gfCNCPoint2[26382] = {X 371.8501, Y 39.8916, Z -3.8333, A 0.000, B 0.000, C 0.000 }
gfCNCPoint2[26383] = {X 370.5669, Y 42.1931, Z -3.8333, A 0.000, B 0.000, C 0.000 }
gfCNCPoint2[26384] = {X 369.0859, Y 44.3727, Z -3.8333, A 0.000, B 0.000, C 0.000 }
gfCNCPoint2[26385] = {X 368.9528, Y 44.5552, Z -3.8333, A 0.000, B 0.000, C 0.000 }
gfCNCPoint2[26386] = {X 368.8456, Y 44.6942, Z -3.8333, A 0.000, B 0.000, C 0.000 }
gfCNCPoint2[26387] = {X 368.1791, Y 45.5125, Z -3.8333, A 0.000, B 0.000, C 0.000 }
gfCNCPoint2[26388] = {X 366.6009, Y 47.2831, Z -3.8333, A 0.000, B 0.000, C 0.000 }
gfCNCPoint2[26389] = {X 364.8716, Y 48.9063, Z -3.8333, A 0.000, B 0.000, C 0.000 }
gfCNCPoint2[26390] = {X 363.0049, Y 50.3694, Z -3.8333, A 0.000, B 0.000, C 0.000 }
gfCNCPoint2[26391] = {X 361.0154, Y 51.6607, Z -3.8333, A 0.000, B 0.000, C 0.000 }
gfCNCPoint2[26392] = {X 358.9191, Y 52.7701, Z -3.8333, A 0.000, B 0.000, C 0.000 }
gfCNCPoint2[26393] = {X 358.4181, Y 53.0061, Z -3.8333, A 0.000, B 0.000, C 0.000 }
gfCNCPoint2[26394] = {X 356.2600, Y 53.8435, Z -3.8333, A 0.000, B 0.000, C 0.000 }
gfCNCPoint2[26395] = {X 354.0408, Y 54.5022, Z -3.8333, A 0.000, B 0.000, C 0.000 }
gfCNCPoint2[26396] = {X 351.7753, Y 54.9779, Z -3.8333, A 0.000, B 0.000, C 0.000 }
gfCNCPoint2[26397] = {X 349.4785, Y 55.2673, Z -3.8333, A 0.000, B 0.000, C 0.000 }
gfCNCPoint2[26398] = {X 347.1658, Y 55.3685, Z -3.8333, A 0.000, B 0.000, C 0.000 }
gfCNCPoint2[26399] = {X 344.5858, Y 55.3167, Z -3.8333, A 0.000, B 0.000, C 0.000 }
gfCNCPoint2[26400] = {X 342.0204, Y 55.0370, Z -3.8333, A 0.000, B 0.000, C 0.000 }
gfCNCPoint2[26401] = {X 339.4898, Y 54.5317, Z -3.8333, A 0.000, B 0.000, C 0.000 }
gfCNCPoint2[26402] = {X 337.0137, Y 53.8047, Z -3.8333, A 0.000, B 0.000, C 0.000 }
gfCNCPoint2[26403] = {X 334.7575, Y 52.9261, Z -3.8333, A 0.000, B 0.000, C 0.000 }
gfCNCPoint2[26404] = {X 332.5819, Y 51.8633, Z -3.8333, A 0.000, B 0.000, C 0.000 }
gfCNCPoint2[26405] = {X 331.5855, Y 51.2776, Z -3.8333, A 0.000, B 0.000, C 0.000 }
gfCNCPoint2[26406] = {X 330.6132, Y 50.6529, Z -3.8333, A 0.000, B 0.000, C 0.000 }
gfCNCPoint2[26407] = {X 331.5791, Y 51.6068, Z -3.8333, A 0.000, B 0.000, C 0.000 }
gfCNCPoint2[26408] = {X 332.4020, Y 52.6865, Z -3.8333, A 0.000, B 0.000, C 0.000 }
gfCNCPoint2[26409] = {X 333.0657, Y 53.8706, Z -3.8333, A 0.000, B 0.000, C 0.000 }
gfCNCPoint2[26410] = {X 333.5573, Y 55.1360, Z -3.8333, A 0.000, B 0.000, C 0.000 }
gfCNCPoint2[26411] = {X 333.8670, Y 56.4577, Z -3.8333, A 0.000, B 0.000, C 0.000 }
gfCNCPoint2[26412] = {X 333.9597, Y 57.2264, Z -3.8333, A 0.000, B 0.000, C 0.000 }
gfCNCPoint2[26413] = {X 333.9907, Y 58.0000, Z -3.8333, A 0.000, B 0.000, C 0.000 }
gfCNCPoint2[26414] = {X 333.9906, Y 58.9572, Z -3.8333, A 0.000, B 0.000, C 0.000 }
gfCNCPoint2[26415] = {X 333.8743, Y 60.4101, Z -3.8333, A 0.000, B 0.000, C 0.000 }
gfCNCPoint2[26416] = {X 333.5421, Y 61.8292, Z -3.8333, A 0.000, B 0.000, C 0.000 }
gfCNCPoint2[26417] = {X 333.0014, Y 63.1827, Z -3.8333, A 0.000, B 0.000, C 0.000 }
gfCNCPoint2[26418] = {X 332.2643, Y 64.4401, Z -3.8333, A 0.000, B 0.000, C 0.000 }
gfCNCPoint2[26419] = {X 331.3475, Y 65.5731, Z -3.8333, A 0.000, B 0.000, C 0.000 }
gfCNCPoint2[26420] = {X 330.2716, Y 66.5563, Z -3.8333, A 0.000, B 0.000, C 0.000 }
gfCNCPoint2[26421] = {X 330.2729, Y 83.2032, Z -3.8333, A 0.000, B 0.000, C 0.000 }
gfCNCPoint2[26422] = {X 330.2766, Y 83.5831, Z -3.8333, A 0.000, B 0.000, C 0.000 }
gfCNCPoint2[26423] = {X 330.3838, Y 83.6086, Z -3.8333, A 0.000, B 0.000, C 0.000 }
gfCNCPoint2[26424] = {X 333.0907, Y 84.1513, Z -3.8333, A 0.000, B 0.000, C 0.000 }
gfCNCPoint2[26425] = {X 335.8298, Y 84.4970, Z -3.8333, A 0.000, B 0.000, C 0.000 }
gfCNCPoint2[26426] = {X 339.8061, Y 84.8050, Z -3.8333, A 0.000, B 0.000, C 0.000 }
gfCNCPoint2[26427] = {X 343.7906, Y 84.9773, Z -3.8333, A 0.000, B 0.000, C 0.000 }
gfCNCPoint2[26428] = {X 347.7787, Y 85.0135, Z -3.8333, A 0.000, B 0.000, C 0.000 }
gfCNCPoint2[26429] = {X 351.9888, Y 84.9781, Z -3.8333, A 0.000, B 0.000, C 0.000 }
gfCNCPoint2[26430] = {X 356.1949, Y 84.7906, Z -3.8333, A 0.000, B 0.000, C 0.000 }
gfCNCPoint2[26431] = {X 360.3914, Y 84.4512, Z -3.8333, A 0.000, B 0.000, C 0.000 }
gfCNCPoint2[26432] = {X 362.9935, Y 84.1044, Z -3.8333, A 0.000, B 0.000, C 0.000 }
gfCNCPoint2[26433] = {X 365.5604, Y 83.5544, Z -3.8333, A 0.000, B 0.000, C 0.000 }
gfCNCPoint2[26434] = {X 365.5591, Y 66.5616, Z -3.8333, A 0.000, B 0.000, C 0.000 }
gfCNCPoint2[26435] = {X 364.4966, Y 65.5962, Z -3.8333, A 0.000, B 0.000, C 0.000 }
gfCNCPoint2[26436] = {X 363.5885, Y 64.4843, Z -3.8333, A 0.000, B 0.000, C 0.000 }
gfCNCPoint2[26437] = {X 362.8549, Y 63.2504, Z -3.8333, A 0.000, B 0.000, C 0.000 }
gfCNCPoint2[26438] = {X 349.9657, Y 69.6713, Z -3.8333, A 0.000, B 0.000, C 0.000 }
gfCNCPoint2[26439] = {X 348.6643, Y 69.7393, Z -3.8333, A 0.000, B 0.000, C 0.000 }
gfCNCPoint2[26440] = {X 347.3614, Y 69.7677, Z -3.8333, A 0.000, B 0.000, C 0.000 }
gfCNCPoint2[26441] = {X 346.5840, Y 69.7768, Z -3.8333, A 0.000, B 0.000, C 0.000 }
gfCNCPoint2[26442] = {X 345.8066, Y 69.7721, Z -3.8333, A 0.000, B 0.000, C 0.000 }
gfCNCPoint2[26443] = {X 345.5899, Y 70.1915, Z -3.8333, A 0.000, B 0.000, C 0.000 }
gfCNCPoint2[26444] = {X 345.3650, Y 70.6066, Z -3.8333, A 0.000, B 0.000, C 0.000 }
gfCNCPoint2[26445] = {X 346.5779, Y 70.6169, Z -3.8333, A 0.000, B 0.000, C 0.000 }
gfCNCPoint2[26446] = {X 347.7907, Y 70.6129, Z -3.8333, A 0.000, B 0.000, C 0.000 }
gfCNCPoint2[26447] = {X 349.1243, Y 70.6187, Z -3.8333, A 0.000, B 0.000, C 0.000 }
gfCNCPoint2[26448] = {X 350.4578, Y 70.6071, Z -3.8333, A 0.000, B 0.000, C 0.000 }
gfCNCPoint2[26449] = {X 350.2066, Y 70.1419, Z -3.8333, A 0.000, B 0.000, C 0.000 }
gfCNCPoint2[26450] = {X 349.9657, Y 69.6713, Z -3.8333, A 0.000, B 0.000, C 0.000 }
gfCNCPoint2[26451] = {X 352.1139, Y 68.6012, Z -3.8333, A 0.000, B 0.000, C 0.000 }
gfCNCPoint2[26452] = {X 351.7677, Y 67.8727, Z -3.8333, A 0.000, B 0.000, C 0.000 }
gfCNCPoint2[26453] = {X 351.4489, Y 67.1318, Z -3.8333, A 0.000, B 0.000, C 0.000 }
gfCNCPoint2[26454] = {X 349.3919, Y 67.3025, Z -3.8333, A 0.000, B 0.000, C 0.000 }
gfCNCPoint2[26455] = {X 347.3288, Y 67.3678, Z -3.8333, A 0.000, B 0.000, C 0.000 }
gfCNCPoint2[26456] = {X 345.8122, Y 67.3719, Z -3.8333, A 0.000, B 0.000, C 0.000 }
gfCNCPoint2[26457] = {X 344.2965, Y 67.3201, Z -3.8333, A 0.000, B 0.000, C 0.000 }
gfCNCPoint2[26458] = {X 343.8102, Y 68.3954, Z -3.8333, A 0.000, B 0.000, C 0.000 }
gfCNCPoint2[26459] = {X 343.2661, Y 69.4427, Z -3.8333, A 0.000, B 0.000, C 0.000 }
gfCNCPoint2[26460] = {X 342.7868, Y 70.2642, Z -3.8333, A 0.000, B 0.000, C 0.000 }
gfCNCPoint2[26461] = {X 342.2719, Y 71.0639, Z -3.8333, A 0.000, B 0.000, C 0.000 }
gfCNCPoint2[26462] = {X 342.2721, Y 72.9175, Z -3.8333, A 0.000, B 0.000, C 0.000 }
gfCNCPoint2[26463] = {X 343.8009, Y 72.9730, Z -3.8333, A 0.000, B 0.000, C 0.000 }
gfCNCPoint2[26464] = {X 345.3303, Y 73.0063, Z -3.8333, A 0.000, B 0.000, C 0.000 }
gfCNCPoint2[26465] = {X 346.5595, Y 73.0169, Z -3.8333, A 0.000, B 0.000, C 0.000 }
gfCNCPoint2[26466] = {X 347.7887, Y 73.0130, Z -3.8333, A 0.000, B 0.000, C 0.000 }
gfCNCPoint2[26467] = {X 349.1416, Y 73.0187, Z -3.8333, A 0.000, B 0.000, C 0.000 }
gfCNCPoint2[26468] = {X 350.4943, Y 73.0069, Z -3.8333, A 0.000, B 0.000, C 0.000 }
gfCNCPoint2[26469] = {X 352.0273, Y 72.9723, Z -3.8333, A 0.000, B 0.000, C 0.000 }
gfCNCPoint2[26470] = {X 353.5596, Y 72.9152, Z -3.8333, A 0.000, B 0.000, C 0.000 }
gfCNCPoint2[26471] = {X 353.5595, Y 71.0777, Z -3.8333, A 0.000, B 0.000, C 0.000 }
gfCNCPoint2[26472] = {X 353.0401, Y 70.2718, Z -3.8333, A 0.000, B 0.000, C 0.000 }
gfCNCPoint2[26473] = {X 352.5569, Y 69.4437, Z -3.8333, A 0.000, B 0.000, C 0.000 }
gfCNCPoint2[26474] = {X 352.3308, Y 69.0249, Z -3.8333, A 0.000, B 0.000, C 0.000 }
gfCNCPoint2[26475] = {X 352.1139, Y 68.6012, Z -3.8333, A 0.000, B 0.000, C 0.000 }
gfCNCPoint2[26476] = {X 354.2621, Y 67.5310, Z -3.8333, A 0.000, B 0.000, C 0.000 }
gfCNCPoint2[26477] = {X 353.5960, Y 66.0387, Z -3.8333, A 0.000, B 0.000, C 0.000 }
gfCNCPoint2[26478] = {X 353.0588, Y 64.4954, Z -3.8333, A 0.000, B 0.000, C 0.000 }
gfCNCPoint2[26479] = {X 350.1865, Y 64.8415, Z -3.8333, A 0.000, B 0.000, C 0.000 }
gfCNCPoint2[26480] = {X 347.2961, Y 64.9680, Z -3.8333, A 0.000, B 0.000, C 0.000 }
gfCNCPoint2[26481] = {X 344.9823, Y 64.9488, Z -3.8333, A 0.000, B 0.000, C 0.000 }
gfCNCPoint2[26482] = {X 342.6738, Y 64.7916, Z -3.8333, A 0.000, B 0.000, C 0.000 }
gfCNCPoint2[26483] = {X 341.9390, Y 66.7265, Z -3.8333, A 0.000, B 0.000, C 0.000 }
gfCNCPoint2[26484] = {X 341.0015, Y 68.5717, Z -3.8333, A 0.000, B 0.000, C 0.000 }
gfCNCPoint2[26485] = {X 339.8719, Y 70.3060, Z -3.8333, A 0.000, B 0.000, C 0.000 }
gfCNCPoint2[26486] = {X 339.8723, Y 75.1904, Z -3.8333, A 0.000, B 0.000, C 0.000 }
gfCNCPoint2[26487] = {X 343.8274, Y 75.3748, Z -3.8333, A 0.000, B 0.000, C 0.000 }
gfCNCPoint2[26488] = {X 347.7867, Y 75.4132, Z -3.8333, A 0.000, B 0.000, C 0.000 }
gfCNCPoint2[26489] = {X 351.8754, Y 75.3776, Z -3.8333, A 0.000, B 0.000, C 0.000 }
gfCNCPoint2[26490] = {X 355.9598, Y 75.1858, Z -3.8333, A 0.000, B 0.000, C 0.000 }
gfCNCPoint2[26491] = {X 355.9594, Y 70.3187, Z -3.8333, A 0.000, B 0.000, C 0.000 }
gfCNCPoint2[26492] = {X 355.0517, Y 68.9608, Z -3.8333, A 0.000, B 0.000, C 0.000 }
gfCNCPoint2[26493] = {X 354.2621, Y 67.5310, Z -3.8333, A 0.000, B 0.000, C 0.000 }
gfCNCPoint2[26494] = {X 356.4103, Y 66.4608, Z -3.8333, A 0.000, B 0.000, C 0.000 }
gfCNCPoint2[26495] = {X 355.7399, Y 64.9296, Z -3.8333, A 0.000, B 0.000, C 0.000 }
gfCNCPoint2[26496] = {X 355.2243, Y 63.3395, Z -3.8333, A 0.000, B 0.000, C 0.000 }
gfCNCPoint2[26497] = {X 354.8685, Y 61.7062, Z -3.8333, A 0.000, B 0.000, C 0.000 }
gfCNCPoint2[26498] = {X 352.3563, Y 62.1755, Z -3.8333, A 0.000, B 0.000, C 0.000 }
gfCNCPoint2[26499] = {X 349.8170, Y 62.4634, Z -3.8333, A 0.000, B 0.000, C 0.000 }
gfCNCPoint2[26500] = {X 347.2635, Y 62.5681, Z -3.8333, A 0.000, B 0.000, C 0.000 }
gfCNCPoint2[26501] = {X 345.1281, Y 62.5526, Z -3.8333, A 0.000, B 0.000, C 0.000 }
gfCNCPoint2[26502] = {X 342.9973, Y 62.4117, Z -3.8333, A 0.000, B 0.000, C 0.000 }
gfCNCPoint2[26503] = {X 340.8785, Y 62.1460, Z -3.8333, A 0.000, B 0.000, C 0.000 }
gfCNCPoint2[26504] = {X 340.4886, Y 63.7339, Z -3.8333, A 0.000, B 0.000, C 0.000 }
gfCNCPoint2[26505] = {X 339.9473, Y 65.2768, Z -3.8333, A 0.000, B 0.000, C 0.000 }
gfCNCPoint2[26506] = {X 339.2595, Y 66.7602, Z -3.8333, A 0.000, B 0.000, C 0.000 }
gfCNCPoint2[26507] = {X 338.4318, Y 68.1703, Z -3.8333, A 0.000, B 0.000, C 0.000 }
gfCNCPoint2[26508] = {X 337.4718, Y 69.4939, Z -3.8333, A 0.000, B 0.000, C 0.000 }
gfCNCPoint2[26509] = {X 337.4724, Y 77.4160, Z -3.8333, A 0.000, B 0.000, C 0.000 }
gfCNCPoint2[26510] = {X 340.9052, Y 77.6563, Z -3.8333, A 0.000, B 0.000, C 0.000 }
gfCNCPoint2[26511] = {X 344.3437, Y 77.7887, Z -3.8333, A 0.000, B 0.000, C 0.000 }
gfCNCPoint2[26512] = {X 347.7847, Y 77.8133, Z -3.8333, A 0.000, B 0.000, C 0.000 }
gfCNCPoint2[26513] = {X 351.3135, Y 77.7924, Z -3.8333, A 0.000, B 0.000, C 0.000 }
gfCNCPoint2[26514] = {X 354.8398, Y 77.6576, Z -3.8333, A 0.000, B 0.000, C 0.000 }
gfCNCPoint2[26515] = {X 358.3599, Y 77.4091, Z -3.8333, A 0.000, B 0.000, C 0.000 }
gfCNCPoint2[26516] = {X 358.3594, Y 69.5053, Z -3.8333, A 0.000, B 0.000, C 0.000 }
gfCNCPoint2[26517] = {X 357.3031, Y 68.0354, Z -3.8333, A 0.000, B 0.000, C 0.000 }
gfCNCPoint2[26518] = {X 356.4103, Y 66.4608, Z -3.8333, A 0.000, B 0.000, C 0.000 }
gfCNCPoint2[26519] = {X 358.5585, Y 65.3907, Z -3.8333, A 0.000, B 0.000, C 0.000 }
gfCNCPoint2[26520] = {X 357.9834, Y 64.0771, Z -3.8333, A 0.000, B 0.000, C 0.000 }
gfCNCPoint2[26521] = {X 357.5411, Y 62.7131, Z -3.8333, A 0.000, B 0.000, C 0.000 }
gfCNCPoint2[26522] = {X 357.2359, Y 61.3120, Z -3.8333, A 0.000, B 0.000, C 0.000 }
gfCNCPoint2[26523] = {X 357.0916, Y 60.1636, Z -3.8333, A 0.000, B 0.000, C 0.000 }
gfCNCPoint2[26524] = {X 357.0395, Y 59.0073, Z -3.8333, A 0.000, B 0.000, C 0.000 }
gfCNCPoint2[26525] = {X 357.0394, Y 58.6392, Z -3.8333, A 0.000, B 0.000, C 0.000 }
gfCNCPoint2[26526] = {X 355.6989, Y 59.0302, Z -3.8333, A 0.000, B 0.000, C 0.000 }
gfCNCPoint2[26527] = {X 354.3432, Y 59.3643, Z -3.8333, A 0.000, B 0.000, C 0.000 }
gfCNCPoint2[26528] = {X 351.9938, Y 59.8031, Z -3.8333, A 0.000, B 0.000, C 0.000 }
gfCNCPoint2[26529] = {X 349.6190, Y 60.0715, Z -3.8333, A 0.000, B 0.000, C 0.000 }
gfCNCPoint2[26530] = {X 347.2310, Y 60.1683, Z -3.8333, A 0.000, B 0.000, C 0.000 }
gfCNCPoint2[26531] = {X 344.3949, Y 60.1141, Z -3.8333, A 0.000, B 0.000, C 0.000 }
gfCNCPoint2[26532] = {X 341.5732, Y 59.8235, Z -3.8333, A 0.000, B 0.000, C 0.000 }
gfCNCPoint2[26533] = {X 338.7856, Y 59.2985, Z -3.8333, A 0.000, B 0.000, C 0.000 }
gfCNCPoint2[26534] = {X 338.6399, Y 60.9979, Z -3.8333, A 0.000, B 0.000, C 0.000 }
gfCNCPoint2[26535] = {X 338.2960, Y 62.6684, Z -3.8333, A 0.000, B 0.000, C 0.000 }
gfCNCPoint2[26536] = {X 337.7585, Y 64.2871, Z -3.8333, A 0.000, B 0.000, C 0.000 }
gfCNCPoint2[26537] = {X 337.0349, Y 65.8316, Z -3.8333, A 0.000, B 0.000, C 0.000 }
gfCNCPoint2[26538] = {X 336.1352, Y 67.2806, Z -3.8333, A 0.000, B 0.000, C 0.000 }
gfCNCPoint2[26539] = {X 335.0717, Y 68.6140, Z -3.8333, A 0.000, B 0.000, C 0.000 }
gfCNCPoint2[26540] = {X 335.0726, Y 79.5885, Z -3.8333, A 0.000, B 0.000, C 0.000 }
gfCNCPoint2[26541] = {X 335.6679, Y 79.6579, Z -3.8333, A 0.000, B 0.000, C 0.000 }
gfCNCPoint2[26542] = {X 336.2643, Y 79.7167, Z -3.8333, A 0.000, B 0.000, C 0.000 }
gfCNCPoint2[26543] = {X 340.0974, Y 80.0139, Z -3.8333, A 0.000, B 0.000, C 0.000 }
gfCNCPoint2[26544] = {X 343.9383, Y 80.1795, Z -3.8333, A 0.000, B 0.000, C 0.000 }
gfCNCPoint2[26545] = {X 347.7827, Y 80.2134, Z -3.8333, A 0.000, B 0.000, C 0.000 }
gfCNCPoint2[26546] = {X 351.8380, Y 80.1804, Z -3.8333, A 0.000, B 0.000, C 0.000 }
gfCNCPoint2[26547] = {X 355.8894, Y 80.0003, Z -3.8333, A 0.000, B 0.000, C 0.000 }
gfCNCPoint2[26548] = {X 359.9315, Y 79.6733, Z -3.8333, A 0.000, B 0.000, C 0.000 }
gfCNCPoint2[26549] = {X 360.3461, Y 79.6317, Z -3.8333, A 0.000, B 0.000, C 0.000 }
gfCNCPoint2[26550] = {X 360.7601, Y 79.5840, Z -3.8333, A 0.000, B 0.000, C 0.000 }
gfCNCPoint2[26551] = {X 360.7593, Y 68.6239, Z -3.8333, A 0.000, B 0.000, C 0.000 }
gfCNCPoint2[26552] = {X 359.9292, Y 67.6140, Z -3.8333, A 0.000, B 0.000, C 0.000 }
gfCNCPoint2[26553] = {X 359.1936, Y 66.5333, Z -3.8333, A 0.000, B 0.000, C 0.000 }
gfCNCPoint2[26554] = {X 358.5585, Y 65.3907, Z -3.8333, A 0.000, B 0.000, C 0.000 }
gfCNCPoint2[26555] = {X 360.7067, Y 64.3205, Z -3.8333, A 0.000, B 0.000, C 0.000 }
gfCNCPoint2[26556] = {X 360.1634, Y 63.0537, Z -3.8333, A 0.000, B 0.000, C 0.000 }
gfCNCPoint2[26557] = {X 359.7680, Y 61.7332, Z -3.8333, A 0.000, B 0.000, C 0.000 }
gfCNCPoint2[26558] = {X 359.5257, Y 60.3762, Z -3.8333, A 0.000, B 0.000, C 0.000 }
gfCNCPoint2[26559] = {X 359.4395, Y 59.0005, Z -3.8333, A 0.000, B 0.000, C 0.000 }
gfCNCPoint2[26560] = {X 359.4393, Y 58.0000, Z -3.8333, A 0.000, B 0.000, C 0.000 }
gfCNCPoint2[26561] = {X 359.5343, Y 56.4880, Z -3.8333, A 0.000, B 0.000, C 0.000 }
gfCNCPoint2[26562] = {X 359.8178, Y 54.9997, Z -3.8333, A 0.000, B 0.000, C 0.000 }
gfCNCPoint2[26563] = {X 359.4090, Y 55.1923, Z -3.8333, A 0.000, B 0.000, C 0.000 }
gfCNCPoint2[26564] = {X 357.8796, Y 55.8125, Z -3.8333, A 0.000, B 0.000, C 0.000 }
gfCNCPoint2[26565] = {X 356.3191, Y 56.3499, Z -3.8333, A 0.000, B 0.000, C 0.000 }
gfCNCPoint2[26566] = {X 354.0855, Y 56.9613, Z -3.8333, A 0.000, B 0.000, C 0.000 }
gfCNCPoint2[26567] = {X 351.8122, Y 57.4030, Z -3.8333, A 0.000, B 0.000, C 0.000 }
gfCNCPoint2[26568] = {X 349.5122, Y 57.6725, Z -3.8333, A 0.000, B 0.000, C 0.000 }
gfCNCPoint2[26569] = {X 347.1984, Y 57.7684, Z -3.8333, A 0.000, B 0.000, C 0.000 }
gfCNCPoint2[26570] = {X 344.5554, Y 57.7194, Z -3.8333, A 0.000, B 0.000, C 0.000 }
gfCNCPoint2[26571] = {X 341.9257, Y 57.4495, Z -3.8333, A 0.000, B 0.000, C 0.000 }
gfCNCPoint2[26572] = {X 339.3279, Y 56.9606, Z -3.8333, A 0.000, B 0.000, C 0.000 }
gfCNCPoint2[26573] = {X 337.7708, Y 56.5573, Z -3.8333, A 0.000, B 0.000, C 0.000 }
gfCNCPoint2[26574] = {X 336.2364, Y 56.0753, Z -3.8333, A 0.000, B 0.000, C 0.000 }
gfCNCPoint2[26575] = {X 336.3520, Y 57.0346, Z -3.8333, A 0.000, B 0.000, C 0.000 }
gfCNCPoint2[26576] = {X 336.3907, Y 58.0000, Z -3.8333, A 0.000, B 0.000, C 0.000 }
gfCNCPoint2[26577] = {X 336.3906, Y 58.9688, Z -3.8333, A 0.000, B 0.000, C 0.000 }
gfCNCPoint2[26578] = {X 336.3892, Y 59.1016, Z -3.8333, A 0.000, B 0.000, C 0.000 }
gfCNCPoint2[26579] = {X 336.3864, Y 59.2343, Z -3.8333, A 0.000, B 0.000, C 0.000 }
gfCNCPoint2[26580] = {X 336.2427, Y 60.7986, Z -3.8333, A 0.000, B 0.000, C 0.000 }
gfCNCPoint2[26581] = {X 335.8980, Y 62.3311, Z -3.8333, A 0.000, B 0.000, C 0.000 }
gfCNCPoint2[26582] = {X 335.3578, Y 63.8062, Z -3.8333, A 0.000, B 0.000, C 0.000 }
gfCNCPoint2[26583] = {X 334.6315, Y 65.1990, Z -3.8333, A 0.000, B 0.000, C 0.000 }
gfCNCPoint2[26584] = {X 333.7310, Y 66.4861, Z -3.8333, A 0.000, B 0.000, C 0.000 }
gfCNCPoint2[26585] = {X 332.6717, Y 67.6460, Z -3.8333, A 0.000, B 0.000, C 0.000 }
gfCNCPoint2[26586] = {X 332.6728, Y 81.6420, Z -3.8333, A 0.000, B 0.000, C 0.000 }
gfCNCPoint2[26587] = {X 334.3529, Y 81.9144, Z -3.8333, A 0.000, B 0.000, C 0.000 }
gfCNCPoint2[26588] = {X 336.0440, Y 82.1065, Z -3.8333, A 0.000, B 0.000, C 0.000 }
gfCNCPoint2[26589] = {X 339.9497, Y 82.4094, Z -3.8333, A 0.000, B 0.000, C 0.000 }
gfCNCPoint2[26590] = {X 343.8635, Y 82.5784, Z -3.8333, A 0.000, B 0.000, C 0.000 }
gfCNCPoint2[26591] = {X 347.7807, Y 82.6135, Z -3.8333, A 0.000, B 0.000, C 0.000 }
gfCNCPoint2[26592] = {X 351.9134, Y 82.5792, Z -3.8333, A 0.000, B 0.000, C 0.000 }
gfCNCPoint2[26593] = {X 356.0420, Y 82.3954, Z -3.8333, A 0.000, B 0.000, C 0.000 }
gfCNCPoint2[26594] = {X 360.1614, Y 82.0623, Z -3.8333, A 0.000, B 0.000, C 0.000 }
gfCNCPoint2[26595] = {X 361.6660, Y 81.8847, Z -3.8333, A 0.000, B 0.000, C 0.000 }
gfCNCPoint2[26596] = {X 363.1603, Y 81.6340, Z -3.8333, A 0.000, B 0.000, C 0.000 }
gfCNCPoint2[26597] = {X 363.1592, Y 67.6539, Z -3.8333, A 0.000, B 0.000, C 0.000 }
gfCNCPoint2[26598] = {X 362.2157, Y 66.6393, Z -3.8333, A 0.000, B 0.000, C 0.000 }
gfCNCPoint2[26599] = {X 361.3946, Y 65.5232, Z -3.8333, A 0.000, B 0.000, C 0.000 }
gfCNCPoint2[26600] = {X 360.7067, Y 64.3205, Z -3.8333, A 0.000, B 0.000, C 0.000 }
gfCNCPoint2[26601] = {X 362.8549, Y 63.2504, Z -3.8333, A 0.000, B 0.000, C 0.000 }
gfCNCPoint2[26602] = {X 362.3011, Y 61.8884, Z -3.8333, A 0.000, B 0.000, C 0.000 }
gfCNCPoint2[26603] = {X 361.9600, Y 60.4583, Z -3.8333, A 0.000, B 0.000, C 0.000 }
gfCNCPoint2[26604] = {X 361.8395, Y 58.9930, Z -3.8333, A 0.000, B 0.000, C 0.000 }
gfCNCPoint2[26605] = {X 361.8393, Y 58.0000, Z -3.8333, A 0.000, B 0.000, C 0.000 }
gfCNCPoint2[26606] = {X 361.9154, Y 56.7884, Z -3.8333, A 0.000, B 0.000, C 0.000 }
gfCNCPoint2[26607] = {X 362.1426, Y 55.5958, Z -3.8333, A 0.000, B 0.000, C 0.000 }
gfCNCPoint2[26608] = {X 362.5739, Y 54.3010, Z -3.8333, A 0.000, B 0.000, C 0.000 }
gfCNCPoint2[26609] = {X 363.1830, Y 53.0798, Z -3.8333, A 0.000, B 0.000, C 0.000 }
gfCNCPoint2[26610] = {X 363.9578, Y 51.9563, Z -3.8333, A 0.000, B 0.000, C 0.000 }
gfCNCPoint2[26611] = {X 364.8829, Y 50.9530, Z -3.8333, A 0.000, B 0.000, C 0.000 }
gfCNCPoint2[26612] = {X 365.9399, Y 50.0897, Z -3.8333, A 0.000, B 0.000, C 0.000 }
gfCNCPoint2[26613] = {X 367.1078, Y 49.3837, Z -3.8333, A 0.000, B 0.000, C 0.000 }
gfCNCPoint2[26614] = {X 368.3634, Y 48.8489, Z -3.8333, A 0.000, B 0.000, C 0.000 }
gfCNCPoint2[26615] = {X 369.6818, Y 48.4960, Z -3.8333, A 0.000, B 0.000, C 0.000 }
gfCNCPoint2[26616] = {X 371.0366, Y 48.3320, Z -3.8333, A 0.000, B 0.000, C 0.000 }
gfCNCPoint2[26617] = {X 371.2779, Y 48.3230, Z -3.8333, A 0.000, B 0.000, C 0.000 }
gfCNCPoint2[26618] = {X 371.5193, Y 48.3200, Z -3.8333, A 0.000, B 0.000, C 0.000 }
gfCNCPoint2[26619] = {X 388.0597, Y 48.3200, Z -3.8333, A 0.000, B 0.000, C 0.000 }
gfCNCPoint2[26620] = {X 389.4419, Y 48.4192, Z -3.8333, A 0.000, B 0.000, C 0.000 }
gfCNCPoint2[26621] = {X 390.7958, Y 48.7147, Z -3.8333, A 0.000, B 0.000, C 0.000 }
gfCNCPoint2[26622] = {X 392.0936, Y 49.2006, Z -3.8333, A 0.000, B 0.000, C 0.000 }
gfCNCPoint2[26623] = {X 393.3087, Y 49.8667, Z -3.8333, A 0.000, B 0.000, C 0.000 }
gfCNCPoint2[26624] = {X 394.5333, Y 49.1962, Z -3.8333, A 0.000, B 0.000, C 0.000 }
gfCNCPoint2[26625] = {X 395.8416, Y 48.7089, Z -3.8333, A 0.000, B 0.000, C 0.000 }
gfCNCPoint2[26626] = {X 397.1858, Y 48.4177, Z -3.8333, A 0.000, B 0.000, C 0.000 }
gfCNCPoint2[26627] = {X 398.5577, Y 48.3200, Z -3.8333, A 0.000, B 0.000, C 0.000 }
gfCNCPoint2[26628] = {X 398.7346, Y 48.3200, Z -3.8333, A 0.000, B 0.000, C 0.000 }
gfCNCPoint2[26629] = {X 398.1859, Y 47.6069, Z -3.8333, A 0.000, B 0.000, C 0.000 }
gfCNCPoint2[26630] = {X 397.7774, Y 46.8051, Z -3.8333, A 0.000, B 0.000, C 0.000 }
gfCNCPoint2[26631] = {X 397.5230, Y 45.9420, Z -3.8333, A 0.000, B 0.000, C 0.000 }
gfCNCPoint2[26632] = {X 397.4561, Y 45.4921, Z -3.8333, A 0.000, B 0.000, C 0.000 }
gfCNCPoint2[26633] = {X 397.4314, Y 45.0378, Z -3.8333, A 0.000, B 0.000, C 0.000 }
gfCNCPoint2[26634] = {X 397.4316, Y 44.1456, Z -3.8333, A 0.000, B 0.000, C 0.000 }
gfCNCPoint2[26635] = {X 397.5413, Y 43.1780, Z -3.8333, A 0.000, B 0.000, C 0.000 }
gfCNCPoint2[26636] = {X 397.8410, Y 42.2514, Z -3.8333, A 0.000, B 0.000, C 0.000 }
gfCNCPoint2[26637] = {X 398.3186, Y 41.4029, Z -3.8333, A 0.000, B 0.000, C 0.000 }
gfCNCPoint2[26638] = {X 398.9552, Y 40.6660, Z -3.8333, A 0.000, B 0.000, C 0.000 }
gfCNCPoint2[26639] = {X 398.9552, Y 31.8228, Z -3.8333, A 0.000, B 0.000, C 0.000 }
gfCNCPoint2[26640] = {X 396.7500, Y 27.9882, Z -3.8333, A 0.000, B 0.000, C 0.000 }
gfCNCPoint2[26641] = {X 386.3474, Y 33.9703, Z -3.8333, A 0.000, B 0.000, C 0.000 }
gfCNCPoint2[26642] = {X 386.2664, Y 34.3979, Z -3.8333, A 0.000, B 0.000, C 0.000 }
gfCNCPoint2[26643] = {X 386.1817, Y 34.8247, Z -3.8333, A 0.000, B 0.000, C 0.000 }
gfCNCPoint2[26644] = {X 386.0227, Y 35.5739, Z -3.8333, A 0.000, B 0.000, C 0.000 }
gfCNCPoint2[26645] = {X 385.8500, Y 36.3200, Z -3.8333, A 0.000, B 0.000, C 0.000 }
gfCNCPoint2[26646] = {X 386.9552, Y 36.3200, Z -3.8333, A 0.000, B 0.000, C 0.000 }
gfCNCPoint2[26647] = {X 386.9552, Y 35.0272, Z -3.8333, A 0.000, B 0.000, C 0.000 }
gfCNCPoint2[26648] = {X 386.3474, Y 33.9703, Z -3.8333, A 0.000, B 0.000, C 0.000 }
gfCNCPoint2[26649] = {X 388.4279, Y 32.7739, Z -3.8333, A 0.000, B 0.000, C 0.000 }
gfCNCPoint2[26650] = {X 384.7446, Y 26.3688, Z -3.8333, A 0.000, B 0.000, C 0.000 }
gfCNCPoint2[26651] = {X 384.6157, Y 28.7693, Z -3.8333, A 0.000, B 0.000, C 0.000 }
gfCNCPoint2[26652] = {X 384.3630, Y 31.1599, Z -3.8333, A 0.000, B 0.000, C 0.000 }
gfCNCPoint2[26653] = {X 383.9874, Y 33.5342, Z -3.8333, A 0.000, B 0.000, C 0.000 }
gfCNCPoint2[26654] = {X 383.9103, Y 33.9411, Z -3.8333, A 0.000, B 0.000, C 0.000 }
gfCNCPoint2[26655] = {X 383.8296, Y 34.3474, Z -3.8333, A 0.000, B 0.000, C 0.000 }
gfCNCPoint2[26656] = {X 383.6797, Y 35.0539, Z -3.8333, A 0.000, B 0.000, C 0.000 }
gfCNCPoint2[26657] = {X 383.5169, Y 35.7576, Z -3.8333, A 0.000, B 0.000, C 0.000 }
gfCNCPoint2[26658] = {X 383.1270, Y 37.2469, Z -3.8333, A 0.000, B 0.000, C 0.000 }
gfCNCPoint2[26659] = {X 382.6793, Y 38.7200, Z -3.8333, A 0.000, B 0.000, C 0.000 }
gfCNCPoint2[26660] = {X 388.0597, Y 38.7200, Z -3.8333, A 0.000, B 0.000, C 0.000 }
gfCNCPoint2[26661] = {X 388.4821, Y 38.7246, Z -3.8333, A 0.000, B 0.000, C 0.000 }
gfCNCPoint2[26662] = {X 388.9043, Y 38.7385, Z -3.8333, A 0.000, B 0.000, C 0.000 }
gfCNCPoint2[26663] = {X 389.1204, Y 38.2363, Z -3.8333, A 0.000, B 0.000, C 0.000 }
gfCNCPoint2[26664] = {X 389.3552, Y 37.7427, Z -3.8333, A 0.000, B 0.000, C 0.000 }
gfCNCPoint2[26665] = {X 389.3552, Y 34.3863, Z -3.8333, A 0.000, B 0.000, C 0.000 }
gfCNCPoint2[26666] = {X 388.4279, Y 32.7739, Z -3.8333, A 0.000, B 0.000, C 0.000 }
gfCNCPoint2[26667] = {X 390.5085, Y 31.5774, Z -3.8333, A 0.000, B 0.000, C 0.000 }
gfCNCPoint2[26668] = {X 386.7859, Y 25.1042, Z -3.8333, A 0.000, B 0.000, C 0.000 }
gfCNCPoint2[26669] = {X 386.1502, Y 24.0176, Z -3.8333, A 0.000, B 0.000, C 0.000 }
gfCNCPoint2[26670] = {X 385.4981, Y 22.9408, Z -3.8333, A 0.000, B 0.000, C 0.000 }
gfCNCPoint2[26671] = {X 384.4697, Y 22.1512, Z -3.8333, A 0.000, B 0.000, C 0.000 }
gfCNCPoint2[26672] = {X 383.5317, Y 21.2559, Z -3.8333, A 0.000, B 0.000, C 0.000 }
gfCNCPoint2[26673] = {X 382.6952, Y 20.2653, Z -3.8333, A 0.000, B 0.000, C 0.000 }
gfCNCPoint2[26674] = {X 381.9696, Y 19.1907, Z -3.8333, A 0.000, B 0.000, C 0.000 }
gfCNCPoint2[26675] = {X 382.2224, Y 21.5532, Z -3.8333, A 0.000, B 0.000, C 0.000 }
gfCNCPoint2[26676] = {X 382.3479, Y 23.9259, Z -3.8333, A 0.000, B 0.000, C 0.000 }
gfCNCPoint2[26677] = {X 382.3456, Y 26.3019, Z -3.8333, A 0.000, B 0.000, C 0.000 }
gfCNCPoint2[26678] = {X 382.2017, Y 28.8399, Z -3.8333, A 0.000, B 0.000, C 0.000 }
gfCNCPoint2[26679] = {X 381.9120, Y 31.3654, Z -3.8333, A 0.000, B 0.000, C 0.000 }
gfCNCPoint2[26680] = {X 381.4776, Y 33.8700, Z -3.8333, A 0.000, B 0.000, C 0.000 }
gfCNCPoint2[26681] = {X 380.9962, Y 35.9392, Z -3.8333, A 0.000, B 0.000, C 0.000 }
gfCNCPoint2[26682] = {X 380.3970, Y 37.9775, Z -3.8333, A 0.000, B 0.000, C 0.000 }
gfCNCPoint2[26683] = {X 379.8415, Y 39.5621, Z -3.8333, A 0.000, B 0.000, C 0.000 }
gfCNCPoint2[26684] = {X 379.2148, Y 41.1200, Z -3.8333, A 0.000, B 0.000, C 0.000 }
gfCNCPoint2[26685] = {X 388.0597, Y 41.1200, Z -3.8333, A 0.000, B 0.000, C 0.000 }
gfCNCPoint2[26686] = {X 389.3256, Y 41.1675, Z -3.8333, A 0.000, B 0.000, C 0.000 }
gfCNCPoint2[26687] = {X 390.5843, Y 41.3099, Z -3.8333, A 0.000, B 0.000, C 0.000 }
gfCNCPoint2[26688] = {X 391.0709, Y 39.7838, Z -3.8333, A 0.000, B 0.000, C 0.000 }
gfCNCPoint2[26689] = {X 391.7552, Y 38.3355, Z -3.8333, A 0.000, B 0.000, C 0.000 }
gfCNCPoint2[26690] = {X 391.7552, Y 33.7454, Z -3.8333, A 0.000, B 0.000, C 0.000 }
gfCNCPoint2[26691] = {X 390.5085, Y 31.5774, Z -3.8333, A 0.000, B 0.000, C 0.000 }
gfCNCPoint2[26692] = {X 392.5890, Y 30.3810, Z -3.8333, A 0.000, B 0.000, C 0.000 }
gfCNCPoint2[26693] = {X 388.8664, Y 23.9077, Z -3.8333, A 0.000, B 0.000, C 0.000 }
gfCNCPoint2[26694] = {X 388.0735, Y 22.5575, Z -3.8333, A 0.000, B 0.000, C 0.000 }
gfCNCPoint2[26695] = {X 387.2562, Y 21.2220, Z -3.8333, A 0.000, B 0.000, C 0.000 }
gfCNCPoint2[26696] = {X 386.3078, Y 20.5569, Z -3.8333, A 0.000, B 0.000, C 0.000 }
gfCNCPoint2[26697] = {X 385.4456, Y 19.7834, Z -3.8333, A 0.000, B 0.000, C 0.000 }
gfCNCPoint2[26698] = {X 384.6820, Y 18.9123, Z -3.8333, A 0.000, B 0.000, C 0.000 }
gfCNCPoint2[26699] = {X 384.0279, Y 17.9564, Z -3.8333, A 0.000, B 0.000, C 0.000 }
gfCNCPoint2[26700] = {X 383.4398, Y 16.8085, Z -3.8333, A 0.000, B 0.000, C 0.000 }
gfCNCPoint2[26701] = {X 383.0094, Y 15.5927, Z -3.8333, A 0.000, B 0.000, C 0.000 }
gfCNCPoint2[26702] = {X 382.7446, Y 14.3305, Z -3.8333, A 0.000, B 0.000, C 0.000 }
gfCNCPoint2[26703] = {X 382.6498, Y 13.0443, Z -3.8333, A 0.000, B 0.000, C 0.000 }
gfCNCPoint2[26704] = {X 382.6496, Y 12.1868, Z -3.8333, A 0.000, B 0.000, C 0.000 }
gfCNCPoint2[26705] = {X 382.6507, Y 12.0459, Z -3.8333, A 0.000, B 0.000, C 0.000 }
gfCNCPoint2[26706] = {X 382.6537, Y 11.9050, Z -3.8333, A 0.000, B 0.000, C 0.000 }
gfCNCPoint2[26707] = {X 377.7925, Y 11.9050, Z -3.8333, A 0.000, B 0.000, C 0.000 }
gfCNCPoint2[26708] = {X 378.4159, Y 13.8446, Z -3.8333, A 0.000, B 0.000, C 0.000 }
gfCNCPoint2[26709] = {X 378.9250, Y 15.8172, Z -3.8333, A 0.000, B 0.000, C 0.000 }
gfCNCPoint2[26710] = {X 379.2995, Y 17.6562, Z -3.8333, A 0.000, B 0.000, C 0.000 }
gfCNCPoint2[26711] = {X 379.5910, Y 19.5101, Z -3.8333, A 0.000, B 0.000, C 0.000 }
gfCNCPoint2[26712] = {X 379.8698, Y 22.2866, Z -3.8333, A 0.000, B 0.000, C 0.000 }
gfCNCPoint2[26713] = {X 379.9627, Y 25.0756, Z -3.8333, A 0.000, B 0.000, C 0.000 }
gfCNCPoint2[26714] = {X 379.8692, Y 27.8646, Z -3.8333, A 0.000, B 0.000, C 0.000 }
gfCNCPoint2[26715] = {X 379.5897, Y 30.6410, Z -3.8333, A 0.000, B 0.000, C 0.000 }
gfCNCPoint2[26716] = {X 379.1255, Y 33.3927, Z -3.8333, A 0.000, B 0.000, C 0.000 }
gfCNCPoint2[26717] = {X 378.5753, Y 35.6997, Z -3.8333, A 0.000, B 0.000, C 0.000 }
gfCNCPoint2[26718] = {X 377.8687, Y 37.9637, Z -3.8333, A 0.000, B 0.000, C 0.000 }
gfCNCPoint2[26719] = {X 377.0090, Y 40.1741, Z -3.8333, A 0.000, B 0.000, C 0.000 }
gfCNCPoint2[26720] = {X 376.2274, Y 41.8693, Z -3.8333, A 0.000, B 0.000, C 0.000 }
gfCNCPoint2[26721] = {X 375.3557, Y 43.5200, Z -3.8333, A 0.000, B 0.000, C 0.000 }
gfCNCPoint2[26722] = {X 388.0597, Y 43.5200, Z -3.8333, A 0.000, B 0.000, C 0.000 }
gfCNCPoint2[26723] = {X 389.6072, Y 43.6029, Z -3.8333, A 0.000, B 0.000, C 0.000 }
gfCNCPoint2[26724] = {X 391.1370, Y 43.8508, Z -3.8333, A 0.000, B 0.000, C 0.000 }
gfCNCPoint2[26725] = {X 392.6316, Y 44.2607, Z -3.8333, A 0.000, B 0.000, C 0.000 }
gfCNCPoint2[26726] = {X 392.7236, Y 42.8756, Z -3.8333, A 0.000, B 0.000, C 0.000 }
gfCNCPoint2[26727] = {X 393.0129, Y 41.5179, Z -3.8333, A 0.000, B 0.000, C 0.000 }
gfCNCPoint2[26728] = {X 393.4934, Y 40.2155, Z -3.8333, A 0.000, B 0.000, C 0.000 }
gfCNCPoint2[26729] = {X 394.1552, Y 38.9952, Z -3.8333, A 0.000, B 0.000, C 0.000 }
gfCNCPoint2[26730] = {X 394.1552, Y 33.1046, Z -3.8333, A 0.000, B 0.000, C 0.000 }
gfCNCPoint2[26731] = {X 392.5890, Y 30.3810, Z -3.8333, A 0.000, B 0.000, C 0.000 }
gfCNCPoint2[26732] = {X 394.6695, Y 29.1846, Z -3.8333, A 0.000, B 0.000, C 0.000 }
gfCNCPoint2[26733] = {X 390.9469, Y 22.7113, Z -3.8333, A 0.000, B 0.000, C 0.000 }
gfCNCPoint2[26734] = {X 390.0888, Y 21.2516, Z -3.8333, A 0.000, B 0.000, C 0.000 }
gfCNCPoint2[26735] = {X 389.2029, Y 19.8087, Z -3.8333, A 0.000, B 0.000, C 0.000 }
gfCNCPoint2[26736] = {X 389.0616, Y 19.6003, Z -3.8333, A 0.000, B 0.000, C 0.000 }
gfCNCPoint2[26737] = {X 388.9057, Y 19.4026, Z -3.8333, A 0.000, B 0.000, C 0.000 }
gfCNCPoint2[26738] = {X 387.8171, Y 18.6908, Z -3.8333, A 0.000, B 0.000, C 0.000 }
gfCNCPoint2[26739] = {X 386.8726, Y 17.7967, Z -3.8333, A 0.000, B 0.000, C 0.000 }
gfCNCPoint2[26740] = {X 386.1023, Y 16.7487, Z -3.8333, A 0.000, B 0.000, C 0.000 }
gfCNCPoint2[26741] = {X 385.5307, Y 15.5805, Z -3.8333, A 0.000, B 0.000, C 0.000 }
gfCNCPoint2[26742] = {X 385.1761, Y 14.3291, Z -3.8333, A 0.000, B 0.000, C 0.000 }
gfCNCPoint2[26743] = {X 385.0498, Y 13.0347, Z -3.8333, A 0.000, B 0.000, C 0.000 }
gfCNCPoint2[26744] = {X 385.0496, Y 12.1868, Z -3.8333, A 0.000, B 0.000, C 0.000 }
gfCNCPoint2[26745] = {X 385.0504, Y 12.0808, Z -3.8333, A 0.000, B 0.000, C 0.000 }
gfCNCPoint2[26746] = {X 385.0527, Y 11.9749, Z -3.8333, A 0.000, B 0.000, C 0.000 }
gfCNCPoint2[26747] = {X 385.1994, Y 10.7177, Z -3.8333, A 0.000, B 0.000, C 0.000 }
gfCNCPoint2[26748] = {X 385.5616, Y 9.5050, Z -3.8333, A 0.000, B 0.000, C 0.000 }
gfCNCPoint2[26749] = {X 374.2010, Y 9.5050, Z -3.8333, A 0.000, B 0.000, C 0.000 }
gfCNCPoint2[26750] = {X 374.9082, Y 11.0877, Z -3.8333, A 0.000, B 0.000, C 0.000 }
gfCNCPoint2[26751] = {X 375.5301, Y 12.7058, Z -3.8333, A 0.000, B 0.000, C 0.000 }
gfCNCPoint2[26752] = {X 376.1105, Y 14.5119, Z -3.8333, A 0.000, B 0.000, C 0.000 }
gfCNCPoint2[26753] = {X 376.5846, Y 16.3488, Z -3.8333, A 0.000, B 0.000, C 0.000 }
gfCNCPoint2[26754] = {X 377.1045, Y 19.0812, Z -3.8333, A 0.000, B 0.000, C 0.000 }
gfCNCPoint2[26755] = {X 377.4302, Y 21.8436, Z -3.8333, A 0.000, B 0.000, C 0.000 }
gfCNCPoint2[26756] = {X 377.5602, Y 24.6220, Z -3.8333, A 0.000, B 0.000, C 0.000 }
gfCNCPoint2[26757] = {X 377.4936, Y 27.4027, Z -3.8333, A 0.000, B 0.000, C 0.000 }
gfCNCPoint2[26758] = {X 377.2310, Y 30.1717, Z -3.8333, A 0.000, B 0.000, C 0.000 }
gfCNCPoint2[26759] = {X 376.7735, Y 32.9153, Z -3.8333, A 0.000, B 0.000, C 0.000 }
gfCNCPoint2[26760] = {X 376.1758, Y 35.3680, Z -3.8333, A 0.000, B 0.000, C 0.000 }
gfCNCPoint2[26761] = {X 375.3884, Y 37.7665, Z -3.8333, A 0.000, B 0.000, C 0.000 }
gfCNCPoint2[26762] = {X 374.4159, Y 40.0961, Z -3.8333, A 0.000, B 0.000, C 0.000 }
gfCNCPoint2[26763] = {X 373.2643, Y 42.3425, Z -3.8333, A 0.000, B 0.000, C 0.000 }
gfCNCPoint2[26764] = {X 372.1961, Y 44.1057, Z -3.8333, A 0.000, B 0.000, C 0.000 }
gfCNCPoint2[26765] = {X 371.0176, Y 45.7970, Z -3.8333, A 0.000, B 0.000, C 0.000 }
gfCNCPoint2[26766] = {X 370.9169, Y 45.9350, Z -3.8333, A 0.000, B 0.000, C 0.000 }
gfCNCPoint2[26767] = {X 371.2180, Y 45.9238, Z -3.8333, A 0.000, B 0.000, C 0.000 }
gfCNCPoint2[26768] = {X 371.5193, Y 45.9200, Z -3.8333, A 0.000, B 0.000, C 0.000 }
gfCNCPoint2[26769] = {X 388.0597, Y 45.9200, Z -3.8333, A 0.000, B 0.000, C 0.000 }
gfCNCPoint2[26770] = {X 389.4143, Y 45.9962, Z -3.8333, A 0.000, B 0.000, C 0.000 }
gfCNCPoint2[26771] = {X 390.7519, Y 46.2238, Z -3.8333, A 0.000, B 0.000, C 0.000 }
gfCNCPoint2[26772] = {X 392.0555, Y 46.6000, Z -3.8333, A 0.000, B 0.000, C 0.000 }
gfCNCPoint2[26773] = {X 393.3087, Y 47.1200, Z -3.8333, A 0.000, B 0.000, C 0.000 }
gfCNCPoint2[26774] = {X 394.2237, Y 46.7243, Z -3.8333, A 0.000, B 0.000, C 0.000 }
gfCNCPoint2[26775] = {X 395.1681, Y 46.4053, Z -3.8333, A 0.000, B 0.000, C 0.000 }
gfCNCPoint2[26776] = {X 395.0678, Y 45.7292, Z -3.8333, A 0.000, B 0.000, C 0.000 }
gfCNCPoint2[26777] = {X 395.0314, Y 45.0468, Z -3.8333, A 0.000, B 0.000, C 0.000 }
gfCNCPoint2[26778] = {X 395.0316, Y 44.1297, Z -3.8333, A 0.000, B 0.000, C 0.000 }
gfCNCPoint2[26779] = {X 395.1397, Y 42.9565, Z -3.8333, A 0.000, B 0.000, C 0.000 }
gfCNCPoint2[26780] = {X 395.4356, Y 41.8161, Z -3.8333, A 0.000, B 0.000, C 0.000 }
gfCNCPoint2[26781] = {X 395.9116, Y 40.7384, Z -3.8333, A 0.000, B 0.000, C 0.000 }
gfCNCPoint2[26782] = {X 396.5552, Y 39.7516, Z -3.8333, A 0.000, B 0.000, C 0.000 }
gfCNCPoint2[26783] = {X 396.5552, Y 32.4637, Z -3.8333, A 0.000, B 0.000, C 0.000 }
gfCNCPoint2[26784] = {X 394.6695, Y 29.1846, Z -3.8333, A 0.000, B 0.000, C 0.000 }
gfCNCPoint2[26785] = {X 396.7500, Y 27.9882, Z -3.8333, A 0.000, B 0.000, C 0.000 }
gfCNCPoint2[26786] = {X 393.0275, Y 21.5149, Z -3.8333, A 0.000, B 0.000, C 0.000 }
gfCNCPoint2[26787] = {X 392.1461, Y 20.0156, Z -3.8333, A 0.000, B 0.000, C 0.000 }
gfCNCPoint2[26788] = {X 391.2361, Y 18.5334, Z -3.8333, A 0.000, B 0.000, C 0.000 }
gfCNCPoint2[26789] = {X 390.8271, Y 17.9602, Z -3.8333, A 0.000, B 0.000, C 0.000 }
gfCNCPoint2[26790] = {X 390.3528, Y 17.4397, Z -3.8333, A 0.000, B 0.000, C 0.000 }
gfCNCPoint2[26791] = {X 389.5427, Y 16.9840, Z -3.8333, A 0.000, B 0.000, C 0.000 }
gfCNCPoint2[26792] = {X 388.8338, Y 16.3830, Z -3.8333, A 0.000, B 0.000, C 0.000 }
gfCNCPoint2[26793] = {X 388.2517, Y 15.6585, Z -3.8333, A 0.000, B 0.000, C 0.000 }
gfCNCPoint2[26794] = {X 387.8175, Y 14.8367, Z -3.8333, A 0.000, B 0.000, C 0.000 }
gfCNCPoint2[26795] = {X 387.5469, Y 13.9476, Z -3.8333, A 0.000, B 0.000, C 0.000 }
gfCNCPoint2[26796] = {X 387.4498, Y 13.0232, Z -3.8333, A 0.000, B 0.000, C 0.000 }
gfCNCPoint2[26797] = {X 387.4496, Y 12.1868, Z -3.8333, A 0.000, B 0.000, C 0.000 }
gfCNCPoint2[26798] = {X 387.5362, Y 11.2717, Z -3.8333, A 0.000, B 0.000, C 0.000 }
gfCNCPoint2[26799] = {X 387.7928, Y 10.3891, Z -3.8333, A 0.000, B 0.000, C 0.000 }
gfCNCPoint2[26800] = {X 388.2375, Y 9.5280, Z -3.8333, A 0.000, B 0.000, C 0.000 }
gfCNCPoint2[26801] = {X 388.8436, Y 8.7718, Z -3.8333, A 0.000, B 0.000, C 0.000 }
gfCNCPoint2[26802] = {X 389.5872, Y 8.1503, Z -3.8333, A 0.000, B 0.000, C 0.000 }
gfCNCPoint2[26803] = {X 390.4390, Y 7.6879, Z -3.8333, A 0.000, B 0.000, C 0.000 }
gfCNCPoint2[26804] = {X 391.3653, Y 7.4030, Z -3.8333, A 0.000, B 0.000, C 0.000 }
gfCNCPoint2[26805] = {X 392.3296, Y 7.3068, Z -3.8333, A 0.000, B 0.000, C 0.000 }
gfCNCPoint2[26806] = {X 399.1118, Y 7.3068, Z -3.8333, A 0.000, B 0.000, C 0.000 }
gfCNCPoint2[26807] = {X 400.0638, Y 7.4006, Z -3.8333, A 0.000, B 0.000, C 0.000 }
gfCNCPoint2[26808] = {X 400.9793, Y 7.6783, Z -3.8333, A 0.000, B 0.000, C 0.000 }
gfCNCPoint2[26809] = {X 401.8229, Y 8.1292, Z -3.8333, A 0.000, B 0.000, C 0.000 }
gfCNCPoint2[26810] = {X 402.5624, Y 8.7361, Z -3.8333, A 0.000, B 0.000, C 0.000 }
gfCNCPoint2[26811] = {X 403.1693, Y 9.4756, Z -3.8333, A 0.000, B 0.000, C 0.000 }
gfCNCPoint2[26812] = {X 403.6203, Y 10.3193, Z -3.8333, A 0.000, B 0.000, C 0.000 }
gfCNCPoint2[26813] = {X 403.8980, Y 11.2348, Z -3.8333, A 0.000, B 0.000, C 0.000 }
gfCNCPoint2[26814] = {X 403.9918, Y 12.1868, Z -3.8333, A 0.000, B 0.000, C 0.000 }
gfCNCPoint2[26815] = {X 403.9915, Y 13.0237, Z -3.8333, A 0.000, B 0.000, C 0.000 }
gfCNCPoint2[26816] = {X 403.9016, Y 13.9115, Z -3.8333, A 0.000, B 0.000, C 0.000 }
gfCNCPoint2[26817] = {X 403.6516, Y 14.7680, Z -3.8333, A 0.000, B 0.000, C 0.000 }
gfCNCPoint2[26818] = {X 405.3650, Y 17.7430, Z -3.8333, A 0.000, B 0.000, C 0.000 }
gfCNCPoint2[26819] = {X 407.2447, Y 14.6981, Z -3.8333, A 0.000, B 0.000, C 0.000 }
gfCNCPoint2[26820] = {X 407.0143, Y 13.8728, Z -3.8333, A 0.000, B 0.000, C 0.000 }
gfCNCPoint2[26821] = {X 406.9317, Y 13.0199, Z -3.8333, A 0.000, B 0.000, C 0.000 }
gfCNCPoint2[26822] = {X 406.9315, Y 12.1868, Z -3.8333, A 0.000, B 0.000, C 0.000 }
gfCNCPoint2[26823] = {X 407.0253, Y 11.2348, Z -3.8333, A 0.000, B 0.000, C 0.000 }
gfCNCPoint2[26824] = {X 407.3030, Y 10.3193, Z -3.8333, A 0.000, B 0.000, C 0.000 }
gfCNCPoint2[26825] = {X 407.7540, Y 9.4756, Z -3.8333, A 0.000, B 0.000, C 0.000 }
gfCNCPoint2[26826] = {X 408.3609, Y 8.7361, Z -3.8333, A 0.000, B 0.000, C 0.000 }
gfCNCPoint2[26827] = {X 409.1004, Y 8.1292, Z -3.8333, A 0.000, B 0.000, C 0.000 }
gfCNCPoint2[26828] = {X 409.9440, Y 7.6783, Z -3.8333, A 0.000, B 0.000, C 0.000 }
gfCNCPoint2[26829] = {X 410.8595, Y 7.4006, Z -3.8333, A 0.000, B 0.000, C 0.000 }
gfCNCPoint2[26830] = {X 411.8115, Y 7.3068, Z -3.8333, A 0.000, B 0.000, C 0.000 }
gfCNCPoint2[26831] = {X 419.3245, Y 7.3068, Z -3.8333, A 0.000, B 0.000, C 0.000 }
gfCNCPoint2[26832] = {X 420.2888, Y 7.4030, Z -3.8333, A 0.000, B 0.000, C 0.000 }
gfCNCPoint2[26833] = {X 421.2151, Y 7.6879, Z -3.8333, A 0.000, B 0.000, C 0.000 }
gfCNCPoint2[26834] = {X 422.0669, Y 8.1503, Z -3.8333, A 0.000, B 0.000, C 0.000 }
gfCNCPoint2[26835] = {X 422.8105, Y 8.7718, Z -3.8333, A 0.000, B 0.000, C 0.000 }
gfCNCPoint2[26836] = {X 423.4166, Y 9.5280, Z -3.8333, A 0.000, B 0.000, C 0.000 }
gfCNCPoint2[26837] = {X 423.8613, Y 10.3891, Z -3.8333, A 0.000, B 0.000, C 0.000 }
gfCNCPoint2[26838] = {X 424.1179, Y 11.2717, Z -3.8333, A 0.000, B 0.000, C 0.000 }
gfCNCPoint2[26839] = {X 424.2045, Y 12.1868, Z -3.8333, A 0.000, B 0.000, C 0.000 }
gfCNCPoint2[26840] = {X 424.2045, Y 12.9780, Z -3.8333, A 0.000, B 0.000, C 0.000 }
gfCNCPoint2[26841] = {X 424.1058, Y 13.9307, Z -3.8333, A 0.000, B 0.000, C 0.000 }
gfCNCPoint2[26842] = {X 423.8253, Y 14.8466, Z -3.8333, A 0.000, B 0.000, C 0.000 }
gfCNCPoint2[26843] = {X 423.3736, Y 15.6912, Z -3.8333, A 0.000, B 0.000, C 0.000 }
gfCNCPoint2[26844] = {X 422.7674, Y 16.4329, Z -3.8333, A 0.000, B 0.000, C 0.000 }
gfCNCPoint2[26845] = {X 422.0296, Y 17.0438, Z -3.8333, A 0.000, B 0.000, C 0.000 }
gfCNCPoint2[26846] = {X 421.1879, Y 17.5010, Z -3.8333, A 0.000, B 0.000, C 0.000 }
gfCNCPoint2[26847] = {X 420.5401, Y 18.3844, Z -3.8333, A 0.000, B 0.000, C 0.000 }
gfCNCPoint2[26848] = {X 419.9509, Y 19.3081, Z -3.8333, A 0.000, B 0.000, C 0.000 }
gfCNCPoint2[26849] = {X 414.1632, Y 28.6173, Z -3.8333, A 0.000, B 0.000, C 0.000 }
gfCNCPoint2[26850] = {X 422.3159, Y 33.6861, Z -3.8333, A 0.000, B 0.000, C 0.000 }
gfCNCPoint2[26851] = {X 421.8913, Y 34.3691, Z -3.8333, A 0.000, B 0.000, C 0.000 }
gfCNCPoint2[26852] = {X 422.1466, Y 34.1004, Z -3.8333, A 0.000, B 0.000, C 0.000 }
gfCNCPoint2[26853] = {X 422.4087, Y 33.8384, Z -3.8333, A 0.000, B 0.000, C 0.000 }
gfCNCPoint2[26854] = {X 422.3622, Y 33.7623, Z -3.8333, A 0.000, B 0.000, C 0.000 }
gfCNCPoint2[26855] = {X 422.3159, Y 33.6861, Z -3.8333, A 0.000, B 0.000, C 0.000 }
gfCNCPoint2[26856] = {X 420.2777, Y 32.4189, Z -3.8333, A 0.000, B 0.000, C 0.000 }
gfCNCPoint2[26857] = {X 419.3068, Y 33.9806, Z -3.8333, A 0.000, B 0.000, C 0.000 }
gfCNCPoint2[26858] = {X 419.3071, Y 38.3389, Z -3.8333, A 0.000, B 0.000, C 0.000 }
gfCNCPoint2[26859] = {X 419.9576, Y 39.7076, Z -3.8333, A 0.000, B 0.000, C 0.000 }
gfCNCPoint2[26860] = {X 420.4333, Y 41.1465, Z -3.8333, A 0.000, B 0.000, C 0.000 }
gfCNCPoint2[26861] = {X 420.6278, Y 41.1585, Z -3.8333, A 0.000, B 0.000, C 0.000 }
gfCNCPoint2[26862] = {X 420.8222, Y 41.1728, Z -3.8333, A 0.000, B 0.000, C 0.000 }
gfCNCPoint2[26863] = {X 421.2842, Y 39.7581, Z -3.8333, A 0.000, B 0.000, C 0.000 }
gfCNCPoint2[26864] = {X 421.9166, Y 38.4111, Z -3.8333, A 0.000, B 0.000, C 0.000 }
gfCNCPoint2[26865] = {X 422.7099, Y 37.1520, Z -3.8333, A 0.000, B 0.000, C 0.000 }
gfCNCPoint2[26866] = {X 423.6520, Y 36.0000, Z -3.8333, A 0.000, B 0.000, C 0.000 }
gfCNCPoint2[26867] = {X 424.3410, Y 35.3138, Z -3.8333, A 0.000, B 0.000, C 0.000 }
gfCNCPoint2[26868] = {X 425.0829, Y 34.6852, Z -3.8333, A 0.000, B 0.000, C 0.000 }
gfCNCPoint2[26869] = {X 425.4261, Y 34.0133, Z -3.8333, A 0.000, B 0.000, C 0.000 }
gfCNCPoint2[26870] = {X 424.8790, Y 33.2426, Z -3.8333, A 0.000, B 0.000, C 0.000 }
gfCNCPoint2[26871] = {X 424.3706, Y 32.4458, Z -3.8333, A 0.000, B 0.000, C 0.000 }
gfCNCPoint2[26872] = {X 423.3898, Y 30.5993, Z -3.8333, A 0.000, B 0.000, C 0.000 }
gfCNCPoint2[26873] = {X 422.6169, Y 28.6566, Z -3.8333, A 0.000, B 0.000, C 0.000 }
gfCNCPoint2[26874] = {X 420.2777, Y 32.4189, Z -3.8333, A 0.000, B 0.000, C 0.000 }
gfCNCPoint2[26875] = {X 418.2396, Y 31.1517, Z -3.8333, A 0.000, B 0.000, C 0.000 }
gfCNCPoint2[26876] = {X 416.9067, Y 33.2954, Z -3.8333, A 0.000, B 0.000, C 0.000 }
gfCNCPoint2[26877] = {X 416.9072, Y 38.9956, Z -3.8333, A 0.000, B 0.000, C 0.000 }
gfCNCPoint2[26878] = {X 417.4885, Y 40.0488, Z -3.8333, A 0.000, B 0.000, C 0.000 }
gfCNCPoint2[26879] = {X 417.9365, Y 41.1652, Z -3.8333, A 0.000, B 0.000, C 0.000 }
gfCNCPoint2[26880] = {X 418.2444, Y 42.3281, Z -3.8333, A 0.000, B 0.000, C 0.000 }
gfCNCPoint2[26881] = {X 418.4076, Y 43.5200, Z -3.8333, A 0.000, B 0.000, C 0.000 }
gfCNCPoint2[26882] = {X 419.4886, Y 43.5200, Z -3.8333, A 0.000, B 0.000, C 0.000 }
gfCNCPoint2[26883] = {X 421.1752, Y 43.6186, Z -3.8333, A 0.000, B 0.000, C 0.000 }
gfCNCPoint2[26884] = {X 422.8389, Y 43.9129, Z -3.8333, A 0.000, B 0.000, C 0.000 }
gfCNCPoint2[26885] = {X 423.0005, Y 42.4234, Z -3.8333, A 0.000, B 0.000, C 0.000 }
gfCNCPoint2[26886] = {X 423.3900, Y 40.9766, Z -3.8333, A 0.000, B 0.000, C 0.000 }
gfCNCPoint2[26887] = {X 423.9980, Y 39.6073, Z -3.8333, A 0.000, B 0.000, C 0.000 }
gfCNCPoint2[26888] = {X 424.8102, Y 38.3482, Z -3.8333, A 0.000, B 0.000, C 0.000 }
gfCNCPoint2[26889] = {X 425.8068, Y 37.2295, Z -3.8333, A 0.000, B 0.000, C 0.000 }
gfCNCPoint2[26890] = {X 426.9642, Y 36.2780, Z -3.8333, A 0.000, B 0.000, C 0.000 }
gfCNCPoint2[26891] = {X 428.2764, Y 33.7096, Z -3.8333, A 0.000, B 0.000, C 0.000 }
gfCNCPoint2[26892] = {X 427.2126, Y 32.3921, Z -3.8333, A 0.000, B 0.000, C 0.000 }
gfCNCPoint2[26893] = {X 426.2879, Y 30.9736, Z -3.8333, A 0.000, B 0.000, C 0.000 }
gfCNCPoint2[26894] = {X 425.5117, Y 29.4687, Z -3.8333, A 0.000, B 0.000, C 0.000 }
gfCNCPoint2[26895] = {X 424.8921, Y 27.8929, Z -3.8333, A 0.000, B 0.000, C 0.000 }
gfCNCPoint2[26896] = {X 424.8101, Y 27.6421, Z -3.8333, A 0.000, B 0.000, C 0.000 }
gfCNCPoint2[26897] = {X 424.7321, Y 27.3901, Z -3.8333, A 0.000, B 0.000, C 0.000 }
gfCNCPoint2[26898] = {X 424.2996, Y 25.6531, Z -3.8333, A 0.000, B 0.000, C 0.000 }
gfCNCPoint2[26899] = {X 424.0101, Y 23.8867, Z -3.8333, A 0.000, B 0.000, C 0.000 }
gfCNCPoint2[26900] = {X 423.8656, Y 22.1025, Z -3.8333, A 0.000, B 0.000, C 0.000 }
gfCNCPoint2[26901] = {X 418.2396, Y 31.1517, Z -3.8333, A 0.000, B 0.000, C 0.000 }
gfCNCPoint2[26902] = {X 416.2014, Y 29.8845, Z -3.8333, A 0.000, B 0.000, C 0.000 }
gfCNCPoint2[26903] = {X 414.5067, Y 32.6103, Z -3.8333, A 0.000, B 0.000, C 0.000 }
gfCNCPoint2[26904] = {X 414.5072, Y 39.7470, Z -3.8333, A 0.000, B 0.000, C 0.000 }
gfCNCPoint2[26905] = {X 415.1558, Y 40.7520, Z -3.8333, A 0.000, B 0.000, C 0.000 }
gfCNCPoint2[26906] = {X 415.6341, Y 41.8483, Z -3.8333, A 0.000, B 0.000, C 0.000 }
gfCNCPoint2[26907] = {X 415.9296, Y 43.0073, Z -3.8333, A 0.000, B 0.000, C 0.000 }
gfCNCPoint2[26908] = {X 416.0347, Y 44.1988, Z -3.8333, A 0.000, B 0.000, C 0.000 }
gfCNCPoint2[26909] = {X 416.0347, Y 44.9999, Z -3.8333, A 0.000, B 0.000, C 0.000 }
gfCNCPoint2[26910] = {X 416.0201, Y 45.4609, Z -3.8333, A 0.000, B 0.000, C 0.000 }
gfCNCPoint2[26911] = {X 415.9763, Y 45.9200, Z -3.8333, A 0.000, B 0.000, C 0.000 }
gfCNCPoint2[26912] = {X 419.4886, Y 45.9200, Z -3.8333, A 0.000, B 0.000, C 0.000 }
gfCNCPoint2[26913] = {X 420.8957, Y 46.0022, Z -3.8333, A 0.000, B 0.000, C 0.000 }
gfCNCPoint2[26914] = {X 422.2836, Y 46.2478, Z -3.8333, A 0.000, B 0.000, C 0.000 }
gfCNCPoint2[26915] = {X 423.4822, Y 46.5992, Z -3.8333, A 0.000, B 0.000, C 0.000 }
gfCNCPoint2[26916] = {X 424.6380, Y 47.0725, Z -3.8333, A 0.000, B 0.000, C 0.000 }
gfCNCPoint2[26917] = {X 425.7388, Y 47.6626, Z -3.8333, A 0.000, B 0.000, C 0.000 }
gfCNCPoint2[26918] = {X 425.4600, Y 46.7984, Z -3.8333, A 0.000, B 0.000, C 0.000 }
gfCNCPoint2[26919] = {X 425.2910, Y 45.9063, Z -3.8333, A 0.000, B 0.000, C 0.000 }
gfCNCPoint2[26920] = {X 425.2344, Y 45.0000, Z -3.8333, A 0.000, B 0.000, C 0.000 }
gfCNCPoint2[26921] = {X 425.2344, Y 44.2090, Z -3.8333, A 0.000, B 0.000, C 0.000 }
gfCNCPoint2[26922] = {X 425.2353, Y 44.0976, Z -3.8333, A 0.000, B 0.000, C 0.000 }
gfCNCPoint2[26923] = {X 425.2378, Y 43.9863, Z -3.8333, A 0.000, B 0.000, C 0.000 }
gfCNCPoint2[26924] = {X 425.3770, Y 42.7748, Z -3.8333, A 0.000, B 0.000, C 0.000 }
gfCNCPoint2[26925] = {X 425.7165, Y 41.6036, Z -3.8333, A 0.000, B 0.000, C 0.000 }
gfCNCPoint2[26926] = {X 426.2468, Y 40.5054, Z -3.8333, A 0.000, B 0.000, C 0.000 }
gfCNCPoint2[26927] = {X 426.9528, Y 39.5112, Z -3.8333, A 0.000, B 0.000, C 0.000 }
gfCNCPoint2[26928] = {X 427.8150, Y 38.6488, Z -3.8333, A 0.000, B 0.000, C 0.000 }
gfCNCPoint2[26929] = {X 428.8090, Y 37.9424, Z -3.8333, A 0.000, B 0.000, C 0.000 }
gfCNCPoint2[26930] = {X 431.2069, Y 33.2486, Z -3.8333, A 0.000, B 0.000, C 0.000 }
gfCNCPoint2[26931] = {X 430.0932, Y 32.1407, Z -3.8333, A 0.000, B 0.000, C 0.000 }
gfCNCPoint2[26932] = {X 429.1078, Y 30.9172, Z -3.8333, A 0.000, B 0.000, C 0.000 }
gfCNCPoint2[26933] = {X 428.2628, Y 29.5929, Z -3.8333, A 0.000, B 0.000, C 0.000 }
gfCNCPoint2[26934] = {X 427.5684, Y 28.1838, Z -3.8333, A 0.000, B 0.000, C 0.000 }
gfCNCPoint2[26935] = {X 427.0329, Y 26.7070, Z -3.8333, A 0.000, B 0.000, C 0.000 }
gfCNCPoint2[26936] = {X 426.6490, Y 25.1628, Z -3.8333, A 0.000, B 0.000, C 0.000 }
gfCNCPoint2[26937] = {X 426.3920, Y 23.5925, Z -3.8333, A 0.000, B 0.000, C 0.000 }
gfCNCPoint2[26938] = {X 426.2637, Y 22.0066, Z -3.8333, A 0.000, B 0.000, C 0.000 }
gfCNCPoint2[26939] = {X 426.2904, Y 19.9403, Z -3.8333, A 0.000, B 0.000, C 0.000 }
gfCNCPoint2[26940] = {X 426.5351, Y 17.8885, Z -3.8333, A 0.000, B 0.000, C 0.000 }
gfCNCPoint2[26941] = {X 426.9953, Y 15.8740, Z -3.8333, A 0.000, B 0.000, C 0.000 }
gfCNCPoint2[26942] = {X 427.6129, Y 14.1182, Z -3.8333, A 0.000, B 0.000, C 0.000 }
gfCNCPoint2[26943] = {X 428.4466, Y 12.4540, Z -3.8333, A 0.000, B 0.000, C 0.000 }
gfCNCPoint2[26944] = {X 429.4832, Y 10.9081, Z -3.8333, A 0.000, B 0.000, C 0.000 }
gfCNCPoint2[26945] = {X 430.7062, Y 9.5050, Z -3.8333, A 0.000, B 0.000, C 0.000 }
gfCNCPoint2[26946] = {X 426.0925, Y 9.5050, Z -3.8333, A 0.000, B 0.000, C 0.000 }
gfCNCPoint2[26947] = {X 426.3754, Y 10.3751, Z -3.8333, A 0.000, B 0.000, C 0.000 }
gfCNCPoint2[26948] = {X 426.5470, Y 11.2737, Z -3.8333, A 0.000, B 0.000, C 0.000 }
gfCNCPoint2[26949] = {X 426.6045, Y 12.1868, Z -3.8333, A 0.000, B 0.000, C 0.000 }
gfCNCPoint2[26950] = {X 426.6045, Y 12.9854, Z -3.8333, A 0.000, B 0.000, C 0.000 }
gfCNCPoint2[26951] = {X 426.4813, Y 14.2872, Z -3.8333, A 0.000, B 0.000, C 0.000 }
gfCNCPoint2[26952] = {X 426.1293, Y 15.5466, Z -3.8333, A 0.000, B 0.000, C 0.000 }
gfCNCPoint2[26953] = {X 425.5596, Y 16.7236, Z -3.8333, A 0.000, B 0.000, C 0.000 }
gfCNCPoint2[26954] = {X 424.7901, Y 17.7809, Z -3.8333, A 0.000, B 0.000, C 0.000 }
gfCNCPoint2[26955] = {X 423.8454, Y 18.6850, Z -3.8333, A 0.000, B 0.000, C 0.000 }
gfCNCPoint2[26956] = {X 422.7553, Y 19.4073, Z -3.8333, A 0.000, B 0.000, C 0.000 }
gfCNCPoint2[26957] = {X 422.3652, Y 19.9717, Z -3.8333, A 0.000, B 0.000, C 0.000 }
gfCNCPoint2[26958] = {X 422.0024, Y 20.5539, Z -3.8333, A 0.000, B 0.000, C 0.000 }
gfCNCPoint2[26959] = {X 416.2014, Y 29.8845, Z -3.8333, A 0.000, B 0.000, C 0.000 }
gfCNCPoint2[26960] = {X 414.1632, Y 28.6173, Z -3.8333, A 0.000, B 0.000, C 0.000 }
gfCNCPoint2[26961] = {X 412.1066, Y 31.9251, Z -3.8333, A 0.000, B 0.000, C 0.000 }
gfCNCPoint2[26962] = {X 412.1073, Y 40.6520, Z -3.8333, A 0.000, B 0.000, C 0.000 }
gfCNCPoint2[26963] = {X 412.7490, Y 41.4085, Z -3.8333, A 0.000, B 0.000, C 0.000 }
gfCNCPoint2[26964] = {X 413.2289, Y 42.2768, Z -3.8333, A 0.000, B 0.000, C 0.000 }
gfCNCPoint2[26965] = {X 413.5280, Y 43.2226, Z -3.8333, A 0.000, B 0.000, C 0.000 }
gfCNCPoint2[26966] = {X 413.6347, Y 44.2089, Z -3.8333, A 0.000, B 0.000, C 0.000 }
gfCNCPoint2[26967] = {X 413.6347, Y 45.0000, Z -3.8333, A 0.000, B 0.000, C 0.000 }
gfCNCPoint2[26968] = {X 413.6249, Y 45.3090, Z -3.8333, A 0.000, B 0.000, C 0.000 }
gfCNCPoint2[26969] = {X 413.5956, Y 45.6167, Z -3.8333, A 0.000, B 0.000, C 0.000 }
gfCNCPoint2[26970] = {X 413.3652, Y 46.5992, Z -3.8333, A 0.000, B 0.000, C 0.000 }
gfCNCPoint2[26971] = {X 412.9377, Y 47.5134, Z -3.8333, A 0.000, B 0.000, C 0.000 }
gfCNCPoint2[26972] = {X 412.3313, Y 48.3200, Z -3.8333, A 0.000, B 0.000, C 0.000 }
gfCNCPoint2[26973] = {X 411.9795, Y 47.9934, Z -3.8333, A 0.000, B 0.000, C 0.000 }
gfCNCPoint2[26974] = {X 411.3003, Y 48.5889, Z -3.8333, A 0.000, B 0.000, C 0.000 }
gfCNCPoint2[26975] = {X 410.5138, Y 49.0331, Z -3.8333, A 0.000, B 0.000, C 0.000 }
gfCNCPoint2[26976] = {X 409.6532, Y 49.3073, Z -3.8333, A 0.000, B 0.000, C 0.000 }
gfCNCPoint2[26977] = {X 408.7547, Y 49.4000, Z -3.8333, A 0.000, B 0.000, C 0.000 }
gfCNCPoint2[26978] = {X 402.3112, Y 49.4000, Z -3.8333, A 0.000, B 0.000, C 0.000 }
gfCNCPoint2[26979] = {X 401.3321, Y 49.2897, Z -3.8333, A 0.000, B 0.000, C 0.000 }
gfCNCPoint2[26980] = {X 400.4021, Y 48.9643, Z -3.8333, A 0.000, B 0.000, C 0.000 }
gfCNCPoint2[26981] = {X 399.5678, Y 48.4400, Z -3.8333, A 0.000, B 0.000, C 0.000 }
gfCNCPoint2[26982] = {X 398.8711, Y 47.7433, Z -3.8333, A 0.000, B 0.000, C 0.000 }
gfCNCPoint2[26983] = {X 398.3469, Y 46.9091, Z -3.8333, A 0.000, B 0.000, C 0.000 }
gfCNCPoint2[26984] = {X 398.0215, Y 45.9791, Z -3.8333, A 0.000, B 0.000, C 0.000 }
gfCNCPoint2[26985] = {X 397.9112, Y 45.0000, Z -3.8333, A 0.000, B 0.000, C 0.000 }
gfCNCPoint2[26986] = {X 397.9116, Y 44.1518, Z -3.8333, A 0.000, B 0.000, C 0.000 }
gfCNCPoint2[26987] = {X 398.0215, Y 43.2300, Z -3.8333, A 0.000, B 0.000, C 0.000 }
gfCNCPoint2[26988] = {X 398.3223, Y 42.3519, Z -3.8333, A 0.000, B 0.000, C 0.000 }
gfCNCPoint2[26989] = {X 398.8006, Y 41.5563, Z -3.8333, A 0.000, B 0.000, C 0.000 }
gfCNCPoint2[26990] = {X 399.4352, Y 40.8789, Z -3.8333, A 0.000, B 0.000, C 0.000 }
gfCNCPoint2[26991] = {X 399.4352, Y 31.6946, Z -3.8333, A 0.000, B 0.000, C 0.000 }
gfCNCPoint2[26992] = {X 393.4436, Y 21.2756, Z -3.8333, A 0.000, B 0.000, C 0.000 }
gfCNCPoint2[26993] = {X 392.5575, Y 19.7684, Z -3.8333, A 0.000, B 0.000, C 0.000 }
gfCNCPoint2[26994] = {X 391.6428, Y 18.2784, Z -3.8333, A 0.000, B 0.000, C 0.000 }
gfCNCPoint2[26995] = {X 391.1721, Y 17.6237, Z -3.8333, A 0.000, B 0.000, C 0.000 }
gfCNCPoint2[26996] = {X 390.6227, Y 17.0334, Z -3.8333, A 0.000, B 0.000, C 0.000 }
gfCNCPoint2[26997] = {X 389.8678, Y 16.6248, Z -3.8333, A 0.000, B 0.000, C 0.000 }
gfCNCPoint2[26998] = {X 389.2066, Y 16.0774, Z -3.8333, A 0.000, B 0.000, C 0.000 }
gfCNCPoint2[26999] = {X 388.6642, Y 15.4121, Z -3.8333, A 0.000, B 0.000, C 0.000 }
gfCNCPoint2[27000] = {X 388.2614, Y 14.6541, Z -3.8333, A 0.000, B 0.000, C 0.000 }
gfCNCPoint2[27001] = {X 388.0133, Y 13.8323, Z -3.8333, A 0.000, B 0.000, C 0.000 }
gfCNCPoint2[27002] = {X 387.9296, Y 12.9779, Z -3.8333, A 0.000, B 0.000, C 0.000 }
gfCNCPoint2[27003] = {X 387.9296, Y 12.1868, Z -3.8333, A 0.000, B 0.000, C 0.000 }
gfCNCPoint2[27004] = {X 388.0399, Y 11.2077, Z -3.8333, A 0.000, B 0.000, C 0.000 }
gfCNCPoint2[27005] = {X 388.3654, Y 10.2777, Z -3.8333, A 0.000, B 0.000, C 0.000 }
gfCNCPoint2[27006] = {X 388.8896, Y 9.4435, Z -3.8333, A 0.000, B 0.000, C 0.000 }
gfCNCPoint2[27007] = {X 389.5863, Y 8.7468, Z -3.8333, A 0.000, B 0.000, C 0.000 }
gfCNCPoint2[27008] = {X 390.4205, Y 8.2226, Z -3.8333, A 0.000, B 0.000, C 0.000 }
gfCNCPoint2[27009] = {X 391.3505, Y 7.8971, Z -3.8333, A 0.000, B 0.000, C 0.000 }
gfCNCPoint2[27010] = {X 392.3296, Y 7.7868, Z -3.8333, A 0.000, B 0.000, C 0.000 }
gfCNCPoint2[27011] = {X 399.1118, Y 7.7868, Z -3.8333, A 0.000, B 0.000, C 0.000 }
gfCNCPoint2[27012] = {X 400.0909, Y 7.8971, Z -3.8333, A 0.000, B 0.000, C 0.000 }
gfCNCPoint2[27013] = {X 401.0208, Y 8.2226, Z -3.8333, A 0.000, B 0.000, C 0.000 }
gfCNCPoint2[27014] = {X 401.8551, Y 8.7468, Z -3.8333, A 0.000, B 0.000, C 0.000 }
gfCNCPoint2[27015] = {X 402.5518, Y 9.4435, Z -3.8333, A 0.000, B 0.000, C 0.000 }
gfCNCPoint2[27016] = {X 403.0760, Y 10.2777, Z -3.8333, A 0.000, B 0.000, C 0.000 }
gfCNCPoint2[27017] = {X 403.4014, Y 11.2077, Z -3.8333, A 0.000, B 0.000, C 0.000 }
gfCNCPoint2[27018] = {X 403.5118, Y 12.1868, Z -3.8333, A 0.000, B 0.000, C 0.000 }
gfCNCPoint2[27019] = {X 403.5115, Y 13.0233, Z -3.8333, A 0.000, B 0.000, C 0.000 }
gfCNCPoint2[27020] = {X 403.4070, Y 13.9326, Z -3.8333, A 0.000, B 0.000, C 0.000 }
gfCNCPoint2[27021] = {X 403.1165, Y 14.8007, Z -3.8333, A 0.000, B 0.000, C 0.000 }
gfCNCPoint2[27022] = {X 405.3506, Y 18.6800, Z -3.8333, A 0.000, B 0.000, C 0.000 }
gfCNCPoint2[27023] = {X 407.7811, Y 14.7431, Z -3.8333, A 0.000, B 0.000, C 0.000 }
gfCNCPoint2[27024] = {X 407.5049, Y 13.8797, Z -3.8333, A 0.000, B 0.000, C 0.000 }
gfCNCPoint2[27025] = {X 407.4115, Y 12.9779, Z -3.8333, A 0.000, B 0.000, C 0.000 }
gfCNCPoint2[27026] = {X 407.4115, Y 12.1868, Z -3.8333, A 0.000, B 0.000, C 0.000 }
gfCNCPoint2[27027] = {X 407.5219, Y 11.2077, Z -3.8333, A 0.000, B 0.000, C 0.000 }
gfCNCPoint2[27028] = {X 407.8473, Y 10.2777, Z -3.8333, A 0.000, B 0.000, C 0.000 }
gfCNCPoint2[27029] = {X 408.3715, Y 9.4435, Z -3.8333, A 0.000, B 0.000, C 0.000 }
gfCNCPoint2[27030] = {X 409.0682, Y 8.7468, Z -3.8333, A 0.000, B 0.000, C 0.000 }
gfCNCPoint2[27031] = {X 409.9024, Y 8.2226, Z -3.8333, A 0.000, B 0.000, C 0.000 }
gfCNCPoint2[27032] = {X 410.8324, Y 7.8971, Z -3.8333, A 0.000, B 0.000, C 0.000 }
gfCNCPoint2[27033] = {X 411.8115, Y 7.7868, Z -3.8333, A 0.000, B 0.000, C 0.000 }
gfCNCPoint2[27034] = {X 419.3245, Y 7.7868, Z -3.8333, A 0.000, B 0.000, C 0.000 }
gfCNCPoint2[27035] = {X 420.3036, Y 7.8971, Z -3.8333, A 0.000, B 0.000, C 0.000 }
gfCNCPoint2[27036] = {X 421.2335, Y 8.2226, Z -3.8333, A 0.000, B 0.000, C 0.000 }
gfCNCPoint2[27037] = {X 422.0678, Y 8.7468, Z -3.8333, A 0.000, B 0.000, C 0.000 }
gfCNCPoint2[27038] = {X 422.7645, Y 9.4435, Z -3.8333, A 0.000, B 0.000, C 0.000 }
gfCNCPoint2[27039] = {X 423.2887, Y 10.2777, Z -3.8333, A 0.000, B 0.000, C 0.000 }
gfCNCPoint2[27040] = {X 423.6141, Y 11.2077, Z -3.8333, A 0.000, B 0.000, C 0.000 }
gfCNCPoint2[27041] = {X 423.7245, Y 12.1868, Z -3.8333, A 0.000, B 0.000, C 0.000 }
gfCNCPoint2[27042] = {X 423.7244, Y 12.9810, Z -3.8333, A 0.000, B 0.000, C 0.000 }
gfCNCPoint2[27043] = {X 423.6304, Y 13.8597, Z -3.8333, A 0.000, B 0.000, C 0.000 }
gfCNCPoint2[27044] = {X 423.3651, Y 14.7028, Z -3.8333, A 0.000, B 0.000, C 0.000 }
gfCNCPoint2[27045] = {X 422.9389, Y 15.4770, Z -3.8333, A 0.000, B 0.000, C 0.000 }
gfCNCPoint2[27046] = {X 422.3686, Y 16.1522, Z -3.8333, A 0.000, B 0.000, C 0.000 }
gfCNCPoint2[27047] = {X 421.6765, Y 16.7018, Z -3.8333, A 0.000, B 0.000, C 0.000 }
gfCNCPoint2[27048] = {X 420.8897, Y 17.1043, Z -3.8333, A 0.000, B 0.000, C 0.000 }
gfCNCPoint2[27049] = {X 420.1827, Y 18.0570, Z -3.8333, A 0.000, B 0.000, C 0.000 }
gfCNCPoint2[27050] = {X 419.5425, Y 19.0559, Z -3.8333, A 0.000, B 0.000, C 0.000 }
gfCNCPoint2[27051] = {X 418.0618, Y 21.4535, Z -3.8333, A 0.000, B 0.000, C 0.000 }
gfCNCPoint2[27052] = {X 411.6266, Y 31.7879, Z -3.8333, A 0.000, B 0.000, C 0.000 }
gfCNCPoint2[27053] = {X 411.6273, Y 40.8619, Z -3.8333, A 0.000, B 0.000, C 0.000 }
gfCNCPoint2[27054] = {X 412.2664, Y 41.5587, Z -3.8333, A 0.000, B 0.000, C 0.000 }
gfCNCPoint2[27055] = {X 412.7466, Y 42.3731, Z -3.8333, A 0.000, B 0.000, C 0.000 }
gfCNCPoint2[27056] = {X 413.0471, Y 43.2695, Z -3.8333, A 0.000, B 0.000, C 0.000 }
gfCNCPoint2[27057] = {X 413.1547, Y 44.2089, Z -3.8333, A 0.000, B 0.000, C 0.000 }
gfCNCPoint2[27058] = {X 413.1545, Y 45.0423, Z -3.8333, A 0.000, B 0.000, C 0.000 }
gfCNCPoint2[27059] = {X 413.0719, Y 45.8494, Z -3.8333, A 0.000, B 0.000, C 0.000 }
gfCNCPoint2[27060] = {X 412.8426, Y 46.6276, Z -3.8333, A 0.000, B 0.000, C 0.000 }
gfCNCPoint2[27061] = {X 412.4743, Y 47.3505, Z -3.8333, A 0.000, B 0.000, C 0.000 }
gfCNCPoint2[27062] = {X 411.9795, Y 47.9934, Z -3.8333, A 0.000, B 0.000, C 0.000 }
gfCNCPoint2[27063] = {X 412.3313, Y 48.3200, Z -3.8333, A 0.000, B 0.000, C 0.000 }
gfCNCPoint2[27064] = {X 419.4886, Y 48.3200, Z -3.8333, A 0.000, B 0.000, C 0.000 }
gfCNCPoint2[27065] = {X 420.8006, Y 48.4093, Z -3.8333, A 0.000, B 0.000, C 0.000 }
gfCNCPoint2[27066] = {X 422.0883, Y 48.6756, Z -3.8333, A 0.000, B 0.000, C 0.000 }
gfCNCPoint2[27067] = {X 423.3281, Y 49.1140, Z -3.8333, A 0.000, B 0.000, C 0.000 }
gfCNCPoint2[27068] = {X 424.4970, Y 49.7164, Z -3.8333, A 0.000, B 0.000, C 0.000 }
gfCNCPoint2[27069] = {X 425.4625, Y 50.3832, Z -3.8333, A 0.000, B 0.000, C 0.000 }
gfCNCPoint2[27070] = {X 426.3402, Y 51.1620, Z -3.8333, A 0.000, B 0.000, C 0.000 }
gfCNCPoint2[27071] = {X 427.1172, Y 52.0412, Z -3.8333, A 0.000, B 0.000, C 0.000 }
gfCNCPoint2[27072] = {X 427.7821, Y 53.0080, Z -3.8333, A 0.000, B 0.000, C 0.000 }
gfCNCPoint2[27073] = {X 428.1268, Y 53.6315, Z -3.8333, A 0.000, B 0.000, C 0.000 }
gfCNCPoint2[27074] = {X 428.4247, Y 54.2786, Z -3.8333, A 0.000, B 0.000, C 0.000 }
gfCNCPoint2[27075] = {X 431.5824, Y 55.5092, Z -3.8333, A 0.000, B 0.000, C 0.000 }
gfCNCPoint2[27076] = {X 439.8778, Y 58.8004, Z -3.8333, A 0.000, B 0.000, C 0.000 }
gfCNCPoint2[27077] = {X 441.6480, Y 54.3388, Z -3.8333, A 0.000, B 0.000, C 0.000 }
gfCNCPoint2[27078] = {X 444.2223, Y 55.3601, Z -3.8333, A 0.000, B 0.000, C 0.000 }
gfCNCPoint2[27079] = {X 444.5425, Y 54.0018, Z -3.8333, A 0.000, B 0.000, C 0.000 }
gfCNCPoint2[27080] = {X 444.9921, Y 52.6806, Z -3.8333, A 0.000, B 0.000, C 0.000 }
gfCNCPoint2[27081] = {X 443.9522, Y 53.3763, Z -3.8333, A 0.000, B 0.000, C 0.000 }
gfCNCPoint2[27082] = {X 442.8313, Y 53.9322, Z -3.8333, A 0.000, B 0.000, C 0.000 }
gfCNCPoint2[27083] = {X 441.6480, Y 54.3388, Z -3.8333, A 0.000, B 0.000, C 0.000 }
gfCNCPoint2[27084] = {X 440.7629, Y 56.5696, Z -3.8333, A 0.000, B 0.000, C 0.000 }
gfCNCPoint2[27085] = {X 446.3797, Y 58.7981, Z -3.8333, A 0.000, B 0.000, C 0.000 }
gfCNCPoint2[27086] = {X 446.3796, Y 58.0000, Z -3.8333, A 0.000, B 0.000, C 0.000 }
gfCNCPoint2[27087] = {X 446.4303, Y 56.8942, Z -3.8333, A 0.000, B 0.000, C 0.000 }
gfCNCPoint2[27088] = {X 446.5821, Y 55.7977, Z -3.8333, A 0.000, B 0.000, C 0.000 }
gfCNCPoint2[27089] = {X 446.8492, Y 54.6645, Z -3.8333, A 0.000, B 0.000, C 0.000 }
gfCNCPoint2[27090] = {X 447.2243, Y 53.5622, Z -3.8333, A 0.000, B 0.000, C 0.000 }
gfCNCPoint2[27091] = {X 447.8767, Y 52.1752, Z -3.8333, A 0.000, B 0.000, C 0.000 }
gfCNCPoint2[27092] = {X 448.6995, Y 50.8820, Z -3.8333, A 0.000, B 0.000, C 0.000 }
gfCNCPoint2[27093] = {X 447.8224, Y 50.1272, Z -3.8333, A 0.000, B 0.000, C 0.000 }
gfCNCPoint2[27094] = {X 447.0760, Y 49.2431, Z -3.8333, A 0.000, B 0.000, C 0.000 }
gfCNCPoint2[27095] = {X 446.4792, Y 48.2518, Z -3.8333, A 0.000, B 0.000, C 0.000 }
gfCNCPoint2[27096] = {X 446.0469, Y 47.1785, Z -3.8333, A 0.000, B 0.000, C 0.000 }
gfCNCPoint2[27097] = {X 445.6333, Y 48.2126, Z -3.8333, A 0.000, B 0.000, C 0.000 }
gfCNCPoint2[27098] = {X 445.0668, Y 49.1715, Z -3.8333, A 0.000, B 0.000, C 0.000 }
gfCNCPoint2[27099] = {X 444.3606, Y 50.0328, Z -3.8333, A 0.000, B 0.000, C 0.000 }
gfCNCPoint2[27100] = {X 443.5314, Y 50.7763, Z -3.8333, A 0.000, B 0.000, C 0.000 }
gfCNCPoint2[27101] = {X 442.7493, Y 51.2996, Z -3.8333, A 0.000, B 0.000, C 0.000 }
gfCNCPoint2[27102] = {X 441.9063, Y 51.7176, Z -3.8333, A 0.000, B 0.000, C 0.000 }
gfCNCPoint2[27103] = {X 441.0164, Y 52.0234, Z -3.8333, A 0.000, B 0.000, C 0.000 }
gfCNCPoint2[27104] = {X 440.0670, Y 52.2156, Z -3.8333, A 0.000, B 0.000, C 0.000 }
gfCNCPoint2[27105] = {X 439.1005, Y 52.2800, Z -3.8333, A 0.000, B 0.000, C 0.000 }
gfCNCPoint2[27106] = {X 432.5144, Y 52.2800, Z -3.8333, A 0.000, B 0.000, C 0.000 }
gfCNCPoint2[27107] = {X 431.6034, Y 52.2228, Z -3.8333, A 0.000, B 0.000, C 0.000 }
gfCNCPoint2[27108] = {X 430.7067, Y 52.0520, Z -3.8333, A 0.000, B 0.000, C 0.000 }
gfCNCPoint2[27109] = {X 429.8384, Y 51.7703, Z -3.8333, A 0.000, B 0.000, C 0.000 }
gfCNCPoint2[27110] = {X 430.0170, Y 52.0773, Z -3.8333, A 0.000, B 0.000, C 0.000 }
gfCNCPoint2[27111] = {X 430.1866, Y 52.3894, Z -3.8333, A 0.000, B 0.000, C 0.000 }
gfCNCPoint2[27112] = {X 432.4642, Y 53.2770, Z -3.8333, A 0.000, B 0.000, C 0.000 }
gfCNCPoint2[27113] = {X 440.7629, Y 56.5696, Z -3.8333, A 0.000, B 0.000, C 0.000 }
gfCNCPoint2[27114] = {X 439.8778, Y 58.8004, Z -3.8333, A 0.000, B 0.000, C 0.000 }
gfCNCPoint2[27115] = {X 449.5096, Y 62.6219, Z -3.8333, A 0.000, B 0.000, C 0.000 }
gfCNCPoint2[27116] = {X 449.1114, Y 61.4469, Z -3.8333, A 0.000, B 0.000, C 0.000 }
gfCNCPoint2[27117] = {X 448.8668, Y 60.2306, Z -3.8333, A 0.000, B 0.000, C 0.000 }
gfCNCPoint2[27118] = {X 448.7798, Y 58.9930, Z -3.8333, A 0.000, B 0.000, C 0.000 }
gfCNCPoint2[27119] = {X 448.7796, Y 58.0000, Z -3.8333, A 0.000, B 0.000, C 0.000 }
gfCNCPoint2[27120] = {X 448.8564, Y 56.7833, Z -3.8333, A 0.000, B 0.000, C 0.000 }
gfCNCPoint2[27121] = {X 449.0855, Y 55.5859, Z -3.8333, A 0.000, B 0.000, C 0.000 }
gfCNCPoint2[27122] = {X 449.4632, Y 54.4268, Z -3.8333, A 0.000, B 0.000, C 0.000 }
gfCNCPoint2[27123] = {X 449.9837, Y 53.3244, Z -3.8333, A 0.000, B 0.000, C 0.000 }
gfCNCPoint2[27124] = {X 450.6386, Y 52.2961, Z -3.8333, A 0.000, B 0.000, C 0.000 }
gfCNCPoint2[27125] = {X 451.3887, Y 51.3890, Z -3.8333, A 0.000, B 0.000, C 0.000 }
gfCNCPoint2[27126] = {X 452.2434, Y 50.5796, Z -3.8333, A 0.000, B 0.000, C 0.000 }
gfCNCPoint2[27127] = {X 453.1901, Y 49.8800, Z -3.8333, A 0.000, B 0.000, C 0.000 }
gfCNCPoint2[27128] = {X 452.3731, Y 49.8442, Z -3.8333, A 0.000, B 0.000, C 0.000 }
gfCNCPoint2[27129] = {X 451.5735, Y 49.6724, Z -3.8333, A 0.000, B 0.000, C 0.000 }
gfCNCPoint2[27130] = {X 450.8138, Y 49.3696, Z -3.8333, A 0.000, B 0.000, C 0.000 }
gfCNCPoint2[27131] = {X 450.1154, Y 48.9441, Z -3.8333, A 0.000, B 0.000, C 0.000 }
gfCNCPoint2[27132] = {X 449.3503, Y 48.2496, Z -3.8333, A 0.000, B 0.000, C 0.000 }
gfCNCPoint2[27133] = {X 448.7486, Y 47.4095, Z -3.8333, A 0.000, B 0.000, C 0.000 }
gfCNCPoint2[27134] = {X 448.3373, Y 46.4616, Z -3.8333, A 0.000, B 0.000, C 0.000 }
gfCNCPoint2[27135] = {X 448.1732, Y 45.7588, Z -3.8333, A 0.000, B 0.000, C 0.000 }
gfCNCPoint2[27136] = {X 448.1146, Y 45.0395, Z -3.8333, A 0.000, B 0.000, C 0.000 }
gfCNCPoint2[27137] = {X 448.1149, Y 44.1417, Z -3.8333, A 0.000, B 0.000, C 0.000 }
gfCNCPoint2[27138] = {X 448.2252, Y 43.1751, Z -3.8333, A 0.000, B 0.000, C 0.000 }
gfCNCPoint2[27139] = {X 448.5250, Y 42.2497, Z -3.8333, A 0.000, B 0.000, C 0.000 }
gfCNCPoint2[27140] = {X 449.0024, Y 41.4021, Z -3.8333, A 0.000, B 0.000, C 0.000 }
gfCNCPoint2[27141] = {X 449.6384, Y 40.6660, Z -3.8333, A 0.000, B 0.000, C 0.000 }
gfCNCPoint2[27142] = {X 449.6384, Y 35.0338, Z -3.8333, A 0.000, B 0.000, C 0.000 }
gfCNCPoint2[27143] = {X 447.8162, Y 35.0338, Z -3.8333, A 0.000, B 0.000, C 0.000 }
gfCNCPoint2[27144] = {X 443.7926, Y 42.8678, Z -3.8333, A 0.000, B 0.000, C 0.000 }
gfCNCPoint2[27145] = {X 443.9302, Y 43.5102, Z -3.8333, A 0.000, B 0.000, C 0.000 }
gfCNCPoint2[27146] = {X 443.9803, Y 44.1653, Z -3.8333, A 0.000, B 0.000, C 0.000 }
gfCNCPoint2[27147] = {X 443.9805, Y 45.0000, Z -3.8333, A 0.000, B 0.000, C 0.000 }
gfCNCPoint2[27148] = {X 443.9242, Y 45.7387, Z -3.8333, A 0.000, B 0.000, C 0.000 }
gfCNCPoint2[27149] = {X 443.7568, Y 46.4603, Z -3.8333, A 0.000, B 0.000, C 0.000 }
gfCNCPoint2[27150] = {X 443.3474, Y 47.4038, Z -3.8333, A 0.000, B 0.000, C 0.000 }
gfCNCPoint2[27151] = {X 442.7493, Y 48.2405, Z -3.8333, A 0.000, B 0.000, C 0.000 }
gfCNCPoint2[27152] = {X 441.9891, Y 48.9332, Z -3.8333, A 0.000, B 0.000, C 0.000 }
gfCNCPoint2[27153] = {X 441.1006, Y 49.4513, Z -3.8333, A 0.000, B 0.000, C 0.000 }
gfCNCPoint2[27154] = {X 440.1232, Y 49.7716, Z -3.8333, A 0.000, B 0.000, C 0.000 }
gfCNCPoint2[27155] = {X 439.1005, Y 49.8800, Z -3.8333, A 0.000, B 0.000, C 0.000 }
gfCNCPoint2[27156] = {X 432.5144, Y 49.8800, Z -3.8333, A 0.000, B 0.000, C 0.000 }
gfCNCPoint2[27157] = {X 431.6014, Y 49.7938, Z -3.8333, A 0.000, B 0.000, C 0.000 }
gfCNCPoint2[27158] = {X 430.7206, Y 49.5383, Z -3.8333, A 0.000, B 0.000, C 0.000 }
gfCNCPoint2[27159] = {X 429.8343, Y 49.0782, Z -3.8333, A 0.000, B 0.000, C 0.000 }
gfCNCPoint2[27160] = {X 429.0603, Y 48.4473, Z -3.8333, A 0.000, B 0.000, C 0.000 }
gfCNCPoint2[27161] = {X 428.4309, Y 47.6720, Z -3.8333, A 0.000, B 0.000, C 0.000 }
gfCNCPoint2[27162] = {X 427.9725, Y 46.7848, Z -3.8333, A 0.000, B 0.000, C 0.000 }
gfCNCPoint2[27163] = {X 427.7197, Y 45.9083, Z -3.8333, A 0.000, B 0.000, C 0.000 }
gfCNCPoint2[27164] = {X 427.6344, Y 45.0000, Z -3.8333, A 0.000, B 0.000, C 0.000 }
gfCNCPoint2[27165] = {X 427.6344, Y 44.2089, Z -3.8333, A 0.000, B 0.000, C 0.000 }
gfCNCPoint2[27166] = {X 427.7263, Y 43.2661, Z -3.8333, A 0.000, B 0.000, C 0.000 }
gfCNCPoint2[27167] = {X 427.9987, Y 42.3588, Z -3.8333, A 0.000, B 0.000, C 0.000 }
gfCNCPoint2[27168] = {X 428.4411, Y 41.5212, Z -3.8333, A 0.000, B 0.000, C 0.000 }
gfCNCPoint2[27169] = {X 429.0371, Y 40.7849, Z -3.8333, A 0.000, B 0.000, C 0.000 }
gfCNCPoint2[27170] = {X 429.7641, Y 40.1776, Z -3.8333, A 0.000, B 0.000, C 0.000 }
gfCNCPoint2[27171] = {X 430.5947, Y 39.7222, Z -3.8333, A 0.000, B 0.000, C 0.000 }
gfCNCPoint2[27172] = {X 434.2533, Y 32.5610, Z -3.8333, A 0.000, B 0.000, C 0.000 }
gfCNCPoint2[27173] = {X 432.9189, Y 31.5582, Z -3.8333, A 0.000, B 0.000, C 0.000 }
gfCNCPoint2[27174] = {X 431.7383, Y 30.3783, Z -3.8333, A 0.000, B 0.000, C 0.000 }
gfCNCPoint2[27175] = {X 430.7346, Y 29.0446, Z -3.8333, A 0.000, B 0.000, C 0.000 }
gfCNCPoint2[27176] = {X 429.9277, Y 27.5834, Z -3.8333, A 0.000, B 0.000, C 0.000 }
gfCNCPoint2[27177] = {X 429.3336, Y 26.0236, Z -3.8333, A 0.000, B 0.000, C 0.000 }
gfCNCPoint2[27178] = {X 428.8995, Y 24.1500, Z -3.8333, A 0.000, B 0.000, C 0.000 }
gfCNCPoint2[27179] = {X 428.6781, Y 22.2397, Z -3.8333, A 0.000, B 0.000, C 0.000 }
gfCNCPoint2[27180] = {X 428.6722, Y 20.3165, Z -3.8333, A 0.000, B 0.000, C 0.000 }
gfCNCPoint2[27181] = {X 428.8818, Y 18.4048, Z -3.8333, A 0.000, B 0.000, C 0.000 }
gfCNCPoint2[27182] = {X 429.3043, Y 16.5286, Z -3.8333, A 0.000, B 0.000, C 0.000 }
gfCNCPoint2[27183] = {X 429.8213, Y 15.0576, Z -3.8333, A 0.000, B 0.000, C 0.000 }
gfCNCPoint2[27184] = {X 430.5196, Y 13.6635, Z -3.8333, A 0.000, B 0.000, C 0.000 }
gfCNCPoint2[27185] = {X 431.3878, Y 12.3684, Z -3.8333, A 0.000, B 0.000, C 0.000 }
gfCNCPoint2[27186] = {X 432.4123, Y 11.1929, Z -3.8333, A 0.000, B 0.000, C 0.000 }
gfCNCPoint2[27187] = {X 433.6945, Y 10.0647, Z -3.8333, A 0.000, B 0.000, C 0.000 }
gfCNCPoint2[27188] = {X 435.1200, Y 9.1242, Z -3.8333, A 0.000, B 0.000, C 0.000 }
gfCNCPoint2[27189] = {X 436.6616, Y 8.3891, Z -3.8333, A 0.000, B 0.000, C 0.000 }
gfCNCPoint2[27190] = {X 438.2899, Y 7.8737, Z -3.8333, A 0.000, B 0.000, C 0.000 }
gfCNCPoint2[27191] = {X 439.9585, Y 7.5564, Z -3.8333, A 0.000, B 0.000, C 0.000 }
gfCNCPoint2[27192] = {X 441.6469, Y 7.3698, Z -3.8333, A 0.000, B 0.000, C 0.000 }
gfCNCPoint2[27193] = {X 443.3446, Y 7.3149, Z -3.8333, A 0.000, B 0.000, C 0.000 }
gfCNCPoint2[27194] = {X 444.0315, Y 7.3109, Z -3.8333, A 0.000, B 0.000, C 0.000 }
gfCNCPoint2[27195] = {X 459.4467, Y 7.3109, Z -3.8333, A 0.000, B 0.000, C 0.000 }
gfCNCPoint2[27196] = {X 460.4095, Y 7.4070, Z -3.8333, A 0.000, B 0.000, C 0.000 }
gfCNCPoint2[27197] = {X 461.3343, Y 7.6915, Z -3.8333, A 0.000, B 0.000, C 0.000 }
gfCNCPoint2[27198] = {X 462.1846, Y 8.1532, Z -3.8333, A 0.000, B 0.000, C 0.000 }
gfCNCPoint2[27199] = {X 462.9269, Y 8.7738, Z -3.8333, A 0.000, B 0.000, C 0.000 }
gfCNCPoint2[27200] = {X 463.5319, Y 9.5289, Z -3.8333, A 0.000, B 0.000, C 0.000 }
gfCNCPoint2[27201] = {X 463.9757, Y 10.3886, Z -3.8333, A 0.000, B 0.000, C 0.000 }
gfCNCPoint2[27202] = {X 464.2316, Y 11.2692, Z -3.8333, A 0.000, B 0.000, C 0.000 }
gfCNCPoint2[27203] = {X 464.3179, Y 12.1822, Z -3.8333, A 0.000, B 0.000, C 0.000 }
gfCNCPoint2[27204] = {X 464.3179, Y 12.9779, Z -3.8333, A 0.000, B 0.000, C 0.000 }
gfCNCPoint2[27205] = {X 464.2174, Y 13.9637, Z -3.8333, A 0.000, B 0.000, C 0.000 }
gfCNCPoint2[27206] = {X 463.9197, Y 14.9089, Z -3.8333, A 0.000, B 0.000, C 0.000 }
gfCNCPoint2[27207] = {X 463.4373, Y 15.7744, Z -3.8333, A 0.000, B 0.000, C 0.000 }
gfCNCPoint2[27208] = {X 462.7899, Y 16.5246, Z -3.8333, A 0.000, B 0.000, C 0.000 }
gfCNCPoint2[27209] = {X 462.7896, Y 16.7698, Z -3.8333, A 0.000, B 0.000, C 0.000 }
gfCNCPoint2[27210] = {X 462.7907, Y 40.6629, Z -3.8333, A 0.000, B 0.000, C 0.000 }
gfCNCPoint2[27211] = {X 463.4317, Y 41.4045, Z -3.8333, A 0.000, B 0.000, C 0.000 }
gfCNCPoint2[27212] = {X 463.9116, Y 42.2592, Z -3.8333, A 0.000, B 0.000, C 0.000 }
gfCNCPoint2[27213] = {X 464.2110, Y 43.1926, Z -3.8333, A 0.000, B 0.000, C 0.000 }
gfCNCPoint2[27214] = {X 464.3178, Y 44.1670, Z -3.8333, A 0.000, B 0.000, C 0.000 }
gfCNCPoint2[27215] = {X 464.3179, Y 45.0000, Z -3.8333, A 0.000, B 0.000, C 0.000 }
gfCNCPoint2[27216] = {X 464.3082, Y 45.3090, Z -3.8333, A 0.000, B 0.000, C 0.000 }
gfCNCPoint2[27217] = {X 464.2788, Y 45.6167, Z -3.8333, A 0.000, B 0.000, C 0.000 }
gfCNCPoint2[27218] = {X 464.0485, Y 46.5992, Z -3.8333, A 0.000, B 0.000, C 0.000 }
gfCNCPoint2[27219] = {X 463.6209, Y 47.5134, Z -3.8333, A 0.000, B 0.000, C 0.000 }
gfCNCPoint2[27220] = {X 463.0145, Y 48.3200, Z -3.8333, A 0.000, B 0.000, C 0.000 }
gfCNCPoint2[27221] = {X 462.6627, Y 47.9934, Z -3.8333, A 0.000, B 0.000, C 0.000 }
gfCNCPoint2[27222] = {X 461.9835, Y 48.5889, Z -3.8333, A 0.000, B 0.000, C 0.000 }
gfCNCPoint2[27223] = {X 461.1970, Y 49.0331, Z -3.8333, A 0.000, B 0.000, C 0.000 }
gfCNCPoint2[27224] = {X 460.3364, Y 49.3073, Z -3.8333, A 0.000, B 0.000, C 0.000 }
gfCNCPoint2[27225] = {X 459.4379, Y 49.4000, Z -3.8333, A 0.000, B 0.000, C 0.000 }
gfCNCPoint2[27226] = {X 452.9945, Y 49.4000, Z -3.8333, A 0.000, B 0.000, C 0.000 }
gfCNCPoint2[27227] = {X 452.0154, Y 49.2897, Z -3.8333, A 0.000, B 0.000, C 0.000 }
gfCNCPoint2[27228] = {X 451.0854, Y 48.9643, Z -3.8333, A 0.000, B 0.000, C 0.000 }
gfCNCPoint2[27229] = {X 450.2511, Y 48.4400, Z -3.8333, A 0.000, B 0.000, C 0.000 }
gfCNCPoint2[27230] = {X 449.5544, Y 47.7433, Z -3.8333, A 0.000, B 0.000, C 0.000 }
gfCNCPoint2[27231] = {X 449.0302, Y 46.9091, Z -3.8333, A 0.000, B 0.000, C 0.000 }
gfCNCPoint2[27232] = {X 448.7048, Y 45.9791, Z -3.8333, A 0.000, B 0.000, C 0.000 }
gfCNCPoint2[27233] = {X 448.5945, Y 45.0000, Z -3.8333, A 0.000, B 0.000, C 0.000 }
gfCNCPoint2[27234] = {X 448.5949, Y 44.1483, Z -3.8333, A 0.000, B 0.000, C 0.000 }
gfCNCPoint2[27235] = {X 448.7053, Y 43.2275, Z -3.8333, A 0.000, B 0.000, C 0.000 }
gfCNCPoint2[27236] = {X 449.0063, Y 42.3503, Z -3.8333, A 0.000, B 0.000, C 0.000 }
gfCNCPoint2[27237] = {X 449.4844, Y 41.5556, Z -3.8333, A 0.000, B 0.000, C 0.000 }
gfCNCPoint2[27238] = {X 450.1184, Y 40.8789, Z -3.8333, A 0.000, B 0.000, C 0.000 }
gfCNCPoint2[27239] = {X 450.1184, Y 34.5538, Z -3.8333, A 0.000, B 0.000, C 0.000 }
gfCNCPoint2[27240] = {X 447.5232, Y 34.5538, Z -3.8333, A 0.000, B 0.000, C 0.000 }
gfCNCPoint2[27241] = {X 443.2763, Y 42.8224, Z -3.8333, A 0.000, B 0.000, C 0.000 }
gfCNCPoint2[27242] = {X 443.4441, Y 43.5066, Z -3.8333, A 0.000, B 0.000, C 0.000 }
gfCNCPoint2[27243] = {X 443.5005, Y 44.2089, Z -3.8333, A 0.000, B 0.000, C 0.000 }
gfCNCPoint2[27244] = {X 443.5005, Y 45.0000, Z -3.8333, A 0.000, B 0.000, C 0.000 }
gfCNCPoint2[27245] = {X 443.3902, Y 45.9791, Z -3.8333, A 0.000, B 0.000, C 0.000 }
gfCNCPoint2[27246] = {X 443.0647, Y 46.9091, Z -3.8333, A 0.000, B 0.000, C 0.000 }
gfCNCPoint2[27247] = {X 442.5405, Y 47.7434, Z -3.8333, A 0.000, B 0.000, C 0.000 }
gfCNCPoint2[27248] = {X 441.8438, Y 48.4401, Z -3.8333, A 0.000, B 0.000, C 0.000 }
gfCNCPoint2[27249] = {X 441.0096, Y 48.9643, Z -3.8333, A 0.000, B 0.000, C 0.000 }
gfCNCPoint2[27250] = {X 440.0796, Y 49.2897, Z -3.8333, A 0.000, B 0.000, C 0.000 }
gfCNCPoint2[27251] = {X 439.1005, Y 49.4000, Z -3.8333, A 0.000, B 0.000, C 0.000 }
gfCNCPoint2[27252] = {X 432.5144, Y 49.4000, Z -3.8333, A 0.000, B 0.000, C 0.000 }
gfCNCPoint2[27253] = {X 431.5353, Y 49.2897, Z -3.8333, A 0.000, B 0.000, C 0.000 }
gfCNCPoint2[27254] = {X 430.6053, Y 48.9643, Z -3.8333, A 0.000, B 0.000, C 0.000 }
gfCNCPoint2[27255] = {X 429.7711, Y 48.4401, Z -3.8333, A 0.000, B 0.000, C 0.000 }
gfCNCPoint2[27256] = {X 429.0743, Y 47.7434, Z -3.8333, A 0.000, B 0.000, C 0.000 }
gfCNCPoint2[27257] = {X 428.5501, Y 46.9091, Z -3.8333, A 0.000, B 0.000, C 0.000 }
gfCNCPoint2[27258] = {X 428.2247, Y 45.9791, Z -3.8333, A 0.000, B 0.000, C 0.000 }
gfCNCPoint2[27259] = {X 428.1144, Y 45.0000, Z -3.8333, A 0.000, B 0.000, C 0.000 }
gfCNCPoint2[27260] = {X 428.1148, Y 44.1483, Z -3.8333, A 0.000, B 0.000, C 0.000 }
gfCNCPoint2[27261] = {X 428.2132, Y 43.2816, Z -3.8333, A 0.000, B 0.000, C 0.000 }
gfCNCPoint2[27262] = {X 428.4806, Y 42.4514, Z -3.8333, A 0.000, B 0.000, C 0.000 }
gfCNCPoint2[27263] = {X 428.9065, Y 41.6903, Z -3.8333, A 0.000, B 0.000, C 0.000 }
gfCNCPoint2[27264] = {X 429.4741, Y 41.0281, Z -3.8333, A 0.000, B 0.000, C 0.000 }
gfCNCPoint2[27265] = {X 430.1613, Y 40.4909, Z -3.8333, A 0.000, B 0.000, C 0.000 }
gfCNCPoint2[27266] = {X 430.9408, Y 40.0998, Z -3.8333, A 0.000, B 0.000, C 0.000 }
gfCNCPoint2[27267] = {X 434.8817, Y 32.3860, Z -3.8333, A 0.000, B 0.000, C 0.000 }
gfCNCPoint2[27268] = {X 433.7182, Y 31.5935, Z -3.8333, A 0.000, B 0.000, C 0.000 }
gfCNCPoint2[27269] = {X 432.6613, Y 30.6635, Z -3.8333, A 0.000, B 0.000, C 0.000 }
gfCNCPoint2[27270] = {X 431.7270, Y 29.6105, Z -3.8333, A 0.000, B 0.000, C 0.000 }
gfCNCPoint2[27271] = {X 430.9296, Y 28.4503, Z -3.8333, A 0.000, B 0.000, C 0.000 }
gfCNCPoint2[27272] = {X 430.2812, Y 27.2007, Z -3.8333, A 0.000, B 0.000, C 0.000 }
gfCNCPoint2[27273] = {X 429.7918, Y 25.8807, Z -3.8333, A 0.000, B 0.000, C 0.000 }
gfCNCPoint2[27274] = {X 429.3712, Y 24.0610, Z -3.8333, A 0.000, B 0.000, C 0.000 }
gfCNCPoint2[27275] = {X 429.1569, Y 22.2057, Z -3.8333, A 0.000, B 0.000, C 0.000 }
gfCNCPoint2[27276] = {X 429.1517, Y 20.3381, Z -3.8333, A 0.000, B 0.000, C 0.000 }
gfCNCPoint2[27277] = {X 429.3556, Y 18.4816, Z -3.8333, A 0.000, B 0.000, C 0.000 }
gfCNCPoint2[27278] = {X 429.7660, Y 16.6596, Z -3.8333, A 0.000, B 0.000, C 0.000 }
gfCNCPoint2[27279] = {X 430.2913, Y 15.1793, Z -3.8333, A 0.000, B 0.000, C 0.000 }
gfCNCPoint2[27280] = {X 431.0074, Y 13.7813, Z -3.8333, A 0.000, B 0.000, C 0.000 }
gfCNCPoint2[27281] = {X 431.9018, Y 12.4901, Z -3.8333, A 0.000, B 0.000, C 0.000 }
gfCNCPoint2[27282] = {X 432.9587, Y 11.3281, Z -3.8333, A 0.000, B 0.000, C 0.000 }
gfCNCPoint2[27283] = {X 434.1597, Y 10.3159, Z -3.8333, A 0.000, B 0.000, C 0.000 }
gfCNCPoint2[27284] = {X 435.4839, Y 9.4710, Z -3.8333, A 0.000, B 0.000, C 0.000 }
gfCNCPoint2[27285] = {X 436.9079, Y 8.8083, Z -3.8333, A 0.000, B 0.000, C 0.000 }
gfCNCPoint2[27286] = {X 438.4070, Y 8.3393, Z -3.8333, A 0.000, B 0.000, C 0.000 }
gfCNCPoint2[27287] = {X 440.0370, Y 8.0300, Z -3.8333, A 0.000, B 0.000, C 0.000 }
gfCNCPoint2[27288] = {X 441.6861, Y 7.8482, Z -3.8333, A 0.000, B 0.000, C 0.000 }
gfCNCPoint2[27289] = {X 443.3444, Y 7.7949, Z -3.8333, A 0.000, B 0.000, C 0.000 }
gfCNCPoint2[27290] = {X 444.0367, Y 7.7909, Z -3.8333, A 0.000, B 0.000, C 0.000 }
gfCNCPoint2[27291] = {X 459.4467, Y 7.7909, Z -3.8333, A 0.000, B 0.000, C 0.000 }
gfCNCPoint2[27292] = {X 460.4238, Y 7.9010, Z -3.8333, A 0.000, B 0.000, C 0.000 }
gfCNCPoint2[27293] = {X 461.3520, Y 8.2258, Z -3.8333, A 0.000, B 0.000, C 0.000 }
gfCNCPoint2[27294] = {X 462.1846, Y 8.7489, Z -3.8333, A 0.000, B 0.000, C 0.000 }
gfCNCPoint2[27295] = {X 462.8799, Y 9.4443, Z -3.8333, A 0.000, B 0.000, C 0.000 }
gfCNCPoint2[27296] = {X 463.4031, Y 10.2769, Z -3.8333, A 0.000, B 0.000, C 0.000 }
gfCNCPoint2[27297] = {X 463.7278, Y 11.2050, Z -3.8333, A 0.000, B 0.000, C 0.000 }
gfCNCPoint2[27298] = {X 463.8379, Y 12.1822, Z -3.8333, A 0.000, B 0.000, C 0.000 }
gfCNCPoint2[27299] = {X 463.8377, Y 13.0201, Z -3.8333, A 0.000, B 0.000, C 0.000 }
gfCNCPoint2[27300] = {X 463.7299, Y 13.9471, Z -3.8333, A 0.000, B 0.000, C 0.000 }
gfCNCPoint2[27301] = {X 463.4290, Y 14.8305, Z -3.8333, A 0.000, B 0.000, C 0.000 }
gfCNCPoint2[27302] = {X 462.9485, Y 15.6305, Z -3.8333, A 0.000, B 0.000, C 0.000 }
gfCNCPoint2[27303] = {X 462.3102, Y 16.3112, Z -3.8333, A 0.000, B 0.000, C 0.000 }
gfCNCPoint2[27304] = {X 462.3096, Y 16.7692, Z -3.8333, A 0.000, B 0.000, C 0.000 }
gfCNCPoint2[27305] = {X 462.3107, Y 40.8761, Z -3.8333, A 0.000, B 0.000, C 0.000 }
gfCNCPoint2[27306] = {X 462.9552, Y 41.5652, Z -3.8333, A 0.000, B 0.000, C 0.000 }
gfCNCPoint2[27307] = {X 463.4380, Y 42.3758, Z -3.8333, A 0.000, B 0.000, C 0.000 }
gfCNCPoint2[27308] = {X 463.7368, Y 43.2708, Z -3.8333, A 0.000, B 0.000, C 0.000 }
gfCNCPoint2[27309] = {X 463.8379, Y 44.2089, Z -3.8333, A 0.000, B 0.000, C 0.000 }
gfCNCPoint2[27310] = {X 463.8379, Y 45.0000, Z -3.8333, A 0.000, B 0.000, C 0.000 }
gfCNCPoint2[27311] = {X 463.7612, Y 45.8182, Z -3.8333, A 0.000, B 0.000, C 0.000 }
gfCNCPoint2[27312] = {X 463.5336, Y 46.6079, Z -3.8333, A 0.000, B 0.000, C 0.000 }
gfCNCPoint2[27313] = {X 463.1632, Y 47.3415, Z -3.8333, A 0.000, B 0.000, C 0.000 }
gfCNCPoint2[27314] = {X 462.6627, Y 47.9934, Z -3.8333, A 0.000, B 0.000, C 0.000 }
gfCNCPoint2[27315] = {X 463.0145, Y 48.3200, Z -3.8333, A 0.000, B 0.000, C 0.000 }
gfCNCPoint2[27316] = {X 472.1884, Y 48.3200, Z -3.8333, A 0.000, B 0.000, C 0.000 }
gfCNCPoint2[27317] = {X 471.5820, Y 47.5134, Z -3.8333, A 0.000, B 0.000, C 0.000 }
gfCNCPoint2[27318] = {X 471.1544, Y 46.5992, Z -3.8333, A 0.000, B 0.000, C 0.000 }
gfCNCPoint2[27319] = {X 470.9241, Y 45.6167, Z -3.8333, A 0.000, B 0.000, C 0.000 }
gfCNCPoint2[27320] = {X 470.8947, Y 45.3090, Z -3.8333, A 0.000, B 0.000, C 0.000 }
gfCNCPoint2[27321] = {X 470.8850, Y 45.0000, Z -3.8333, A 0.000, B 0.000, C 0.000 }
gfCNCPoint2[27322] = {X 470.8850, Y 44.2089, Z -3.8333, A 0.000, B 0.000, C 0.000 }
gfCNCPoint2[27323] = {X 470.9769, Y 43.2661, Z -3.8333, A 0.000, B 0.000, C 0.000 }
gfCNCPoint2[27324] = {X 471.2492, Y 42.3588, Z -3.8333, A 0.000, B 0.000, C 0.000 }
gfCNCPoint2[27325] = {X 471.6917, Y 41.5212, Z -3.8333, A 0.000, B 0.000, C 0.000 }
gfCNCPoint2[27326] = {X 472.2877, Y 40.7849, Z -3.8333, A 0.000, B 0.000, C 0.000 }
gfCNCPoint2[27327] = {X 473.0147, Y 40.1776, Z -3.8333, A 0.000, B 0.000, C 0.000 }
gfCNCPoint2[27328] = {X 473.8453, Y 39.7222, Z -3.8333, A 0.000, B 0.000, C 0.000 }
gfCNCPoint2[27329] = {X 477.5003, Y 32.5678, Z -3.8333, A 0.000, B 0.000, C 0.000 }
gfCNCPoint2[27330] = {X 476.2830, Y 31.6578, Z -3.8333, A 0.000, B 0.000, C 0.000 }
gfCNCPoint2[27331] = {X 475.1902, Y 30.6015, Z -3.8333, A 0.000, B 0.000, C 0.000 }
gfCNCPoint2[27332] = {X 474.2393, Y 29.4159, Z -3.8333, A 0.000, B 0.000, C 0.000 }
gfCNCPoint2[27333] = {X 473.4454, Y 28.1198, Z -3.8333, A 0.000, B 0.000, C 0.000 }
gfCNCPoint2[27334] = {X 472.8213, Y 26.7340, Z -3.8333, A 0.000, B 0.000, C 0.000 }
gfCNCPoint2[27335] = {X 472.3770, Y 25.2806, Z -3.8333, A 0.000, B 0.000, C 0.000 }
gfCNCPoint2[27336] = {X 472.0532, Y 23.5414, Z -3.8333, A 0.000, B 0.000, C 0.000 }
gfCNCPoint2[27337] = {X 471.9085, Y 21.7782, Z -3.8333, A 0.000, B 0.000, C 0.000 }
gfCNCPoint2[27338] = {X 471.9444, Y 20.0095, Z -3.8333, A 0.000, B 0.000, C 0.000 }
gfCNCPoint2[27339] = {X 472.1605, Y 18.2537, Z -3.8333, A 0.000, B 0.000, C 0.000 }
gfCNCPoint2[27340] = {X 472.5546, Y 16.5291, Z -3.8333, A 0.000, B 0.000, C 0.000 }
gfCNCPoint2[27341] = {X 473.0732, Y 15.0581, Z -3.8333, A 0.000, B 0.000, C 0.000 }
gfCNCPoint2[27342] = {X 473.7724, Y 13.6638, Z -3.8333, A 0.000, B 0.000, C 0.000 }
gfCNCPoint2[27343] = {X 474.6414, Y 12.3685, Z -3.8333, A 0.000, B 0.000, C 0.000 }
gfCNCPoint2[27344] = {X 475.6661, Y 11.1926, Z -3.8333, A 0.000, B 0.000, C 0.000 }
gfCNCPoint2[27345] = {X 476.7437, Y 10.2235, Z -3.8333, A 0.000, B 0.000, C 0.000 }
gfCNCPoint2[27346] = {X 477.9270, Y 9.3869, Z -3.8333, A 0.000, B 0.000, C 0.000 }
gfCNCPoint2[27347] = {X 479.1999, Y 8.6942, Z -3.8333, A 0.000, B 0.000, C 0.000 }
gfCNCPoint2[27348] = {X 480.5449, Y 8.1549, Z -3.8333, A 0.000, B 0.000, C 0.000 }
gfCNCPoint2[27349] = {X 481.9438, Y 7.7763, Z -3.8333, A 0.000, B 0.000, C 0.000 }
gfCNCPoint2[27350] = {X 484.0949, Y 7.4409, Z -3.8333, A 0.000, B 0.000, C 0.000 }
gfCNCPoint2[27351] = {X 486.2688, Y 7.3231, Z -3.8333, A 0.000, B 0.000, C 0.000 }
gfCNCPoint2[27352] = {X 486.9707, Y 7.3109, Z -3.8333, A 0.000, B 0.000, C 0.000 }
gfCNCPoint2[27353] = {X 502.2122, Y 7.3109, Z -3.8333, A 0.000, B 0.000, C 0.000 }
gfCNCPoint2[27354] = {X 502.7438, Y 7.3151, Z -3.8333, A 0.000, B 0.000, C 0.000 }
gfCNCPoint2[27355] = {X 503.6980, Y 7.4172, Z -3.8333, A 0.000, B 0.000, C 0.000 }
gfCNCPoint2[27356] = {X 504.6137, Y 7.7048, Z -3.8333, A 0.000, B 0.000, C 0.000 }
gfCNCPoint2[27357] = {X 505.4550, Y 8.1667, Z -3.8333, A 0.000, B 0.000, C 0.000 }
gfCNCPoint2[27358] = {X 506.1892, Y 8.7848, Z -3.8333, A 0.000, B 0.000, C 0.000 }
gfCNCPoint2[27359] = {X 506.7877, Y 9.5350, Z -3.8333, A 0.000, B 0.000, C 0.000 }
gfCNCPoint2[27360] = {X 507.2273, Y 10.3882, Z -3.8333, A 0.000, B 0.000, C 0.000 }
gfCNCPoint2[27361] = {X 507.4824, Y 11.2668, Z -3.8333, A 0.000, B 0.000, C 0.000 }
gfCNCPoint2[27362] = {X 507.5685, Y 12.1776, Z -3.8333, A 0.000, B 0.000, C 0.000 }
gfCNCPoint2[27363] = {X 507.5683, Y 13.0237, Z -3.8333, A 0.000, B 0.000, C 0.000 }
gfCNCPoint2[27364] = {X 507.4609, Y 13.9972, Z -3.8333, A 0.000, B 0.000, C 0.000 }
gfCNCPoint2[27365] = {X 507.1613, Y 14.9296, Z -3.8333, A 0.000, B 0.000, C 0.000 }
gfCNCPoint2[27366] = {X 506.6815, Y 15.7834, Z -3.8333, A 0.000, B 0.000, C 0.000 }
gfCNCPoint2[27367] = {X 506.0409, Y 16.5243, Z -3.8333, A 0.000, B 0.000, C 0.000 }
gfCNCPoint2[27368] = {X 506.0408, Y 40.6625, Z -3.8333, A 0.000, B 0.000, C 0.000 }
gfCNCPoint2[27369] = {X 506.6819, Y 41.4040, Z -3.8333, A 0.000, B 0.000, C 0.000 }
gfCNCPoint2[27370] = {X 507.1619, Y 42.2587, Z -3.8333, A 0.000, B 0.000, C 0.000 }
gfCNCPoint2[27371] = {X 507.4614, Y 43.1921, Z -3.8333, A 0.000, B 0.000, C 0.000 }
gfCNCPoint2[27372] = {X 507.5683, Y 44.1665, Z -3.8333, A 0.000, B 0.000, C 0.000 }
gfCNCPoint2[27373] = {X 507.5685, Y 45.0000, Z -3.8333, A 0.000, B 0.000, C 0.000 }
gfCNCPoint2[27374] = {X 507.4747, Y 45.9520, Z -3.8333, A 0.000, B 0.000, C 0.000 }
gfCNCPoint2[27375] = {X 507.1970, Y 46.8675, Z -3.8333, A 0.000, B 0.000, C 0.000 }
gfCNCPoint2[27376] = {X 506.7461, Y 47.7112, Z -3.8333, A 0.000, B 0.000, C 0.000 }
gfCNCPoint2[27377] = {X 506.1392, Y 48.4507, Z -3.8333, A 0.000, B 0.000, C 0.000 }
gfCNCPoint2[27378] = {X 505.3997, Y 49.0576, Z -3.8333, A 0.000, B 0.000, C 0.000 }
gfCNCPoint2[27379] = {X 504.5560, Y 49.5085, Z -3.8333, A 0.000, B 0.000, C 0.000 }
gfCNCPoint2[27380] = {X 503.6405, Y 49.7862, Z -3.8333, A 0.000, B 0.000, C 0.000 }
gfCNCPoint2[27381] = {X 502.6885, Y 49.8800, Z -3.8333, A 0.000, B 0.000, C 0.000 }
gfCNCPoint2[27382] = {X 496.2450, Y 49.8800, Z -3.8333, A 0.000, B 0.000, C 0.000 }
gfCNCPoint2[27383] = {X 495.2220, Y 49.7716, Z -3.8333, A 0.000, B 0.000, C 0.000 }
gfCNCPoint2[27384] = {X 494.2445, Y 49.4511, Z -3.8333, A 0.000, B 0.000, C 0.000 }
gfCNCPoint2[27385] = {X 493.3559, Y 48.9328, Z -3.8333, A 0.000, B 0.000, C 0.000 }
gfCNCPoint2[27386] = {X 492.5956, Y 48.2398, Z -3.8333, A 0.000, B 0.000, C 0.000 }
gfCNCPoint2[27387] = {X 491.9976, Y 47.4028, Z -3.8333, A 0.000, B 0.000, C 0.000 }
gfCNCPoint2[27388] = {X 491.5882, Y 46.4590, Z -3.8333, A 0.000, B 0.000, C 0.000 }
gfCNCPoint2[27389] = {X 491.4241, Y 45.7570, Z -3.8333, A 0.000, B 0.000, C 0.000 }
gfCNCPoint2[27390] = {X 491.3652, Y 45.0385, Z -3.8333, A 0.000, B 0.000, C 0.000 }
gfCNCPoint2[27391] = {X 491.3655, Y 44.1416, Z -3.8333, A 0.000, B 0.000, C 0.000 }
gfCNCPoint2[27392] = {X 491.4758, Y 43.1751, Z -3.8333, A 0.000, B 0.000, C 0.000 }
gfCNCPoint2[27393] = {X 491.7756, Y 42.2496, Z -3.8333, A 0.000, B 0.000, C 0.000 }
gfCNCPoint2[27394] = {X 492.2530, Y 41.4020, Z -3.8333, A 0.000, B 0.000, C 0.000 }
gfCNCPoint2[27395] = {X 492.8890, Y 40.6660, Z -3.8333, A 0.000, B 0.000, C 0.000 }
gfCNCPoint2[27396] = {X 492.8890, Y 35.0338, Z -3.8333, A 0.000, B 0.000, C 0.000 }
gfCNCPoint2[27397] = {X 491.0661, Y 35.0338, Z -3.8333, A 0.000, B 0.000, C 0.000 }
gfCNCPoint2[27398] = {X 487.0431, Y 42.8678, Z -3.8333, A 0.000, B 0.000, C 0.000 }
gfCNCPoint2[27399] = {X 487.1807, Y 43.5100, Z -3.8333, A 0.000, B 0.000, C 0.000 }
gfCNCPoint2[27400] = {X 487.2308, Y 44.1648, Z -3.8333, A 0.000, B 0.000, C 0.000 }
gfCNCPoint2[27401] = {X 487.2310, Y 45.0000, Z -3.8333, A 0.000, B 0.000, C 0.000 }
gfCNCPoint2[27402] = {X 487.1749, Y 45.7380, Z -3.8333, A 0.000, B 0.000, C 0.000 }
gfCNCPoint2[27403] = {X 487.0078, Y 46.4590, Z -3.8333, A 0.000, B 0.000, C 0.000 }
gfCNCPoint2[27404] = {X 486.5939, Y 47.4110, Z -3.8333, A 0.000, B 0.000, C 0.000 }
gfCNCPoint2[27405] = {X 485.9879, Y 48.2538, Z -3.8333, A 0.000, B 0.000, C 0.000 }
gfCNCPoint2[27406] = {X 485.2175, Y 48.9494, Z -3.8333, A 0.000, B 0.000, C 0.000 }
gfCNCPoint2[27407] = {X 484.3173, Y 49.4663, Z -3.8333, A 0.000, B 0.000, C 0.000 }
gfCNCPoint2[27408] = {X 483.3557, Y 49.7755, Z -3.8333, A 0.000, B 0.000, C 0.000 }
gfCNCPoint2[27409] = {X 482.3510, Y 49.8800, Z -3.8333, A 0.000, B 0.000, C 0.000 }
gfCNCPoint2[27410] = {X 480.2695, Y 49.8800, Z -3.8333, A 0.000, B 0.000, C 0.000 }
gfCNCPoint2[27411] = {X 480.2695, Y 49.4000, Z -3.8333, A 0.000, B 0.000, C 0.000 }
gfCNCPoint2[27412] = {X 475.7650, Y 49.4000, Z -3.8333, A 0.000, B 0.000, C 0.000 }
gfCNCPoint2[27413] = {X 474.7859, Y 49.2897, Z -3.8333, A 0.000, B 0.000, C 0.000 }
gfCNCPoint2[27414] = {X 473.8559, Y 48.9643, Z -3.8333, A 0.000, B 0.000, C 0.000 }
gfCNCPoint2[27415] = {X 473.0216, Y 48.4401, Z -3.8333, A 0.000, B 0.000, C 0.000 }
gfCNCPoint2[27416] = {X 472.3249, Y 47.7434, Z -3.8333, A 0.000, B 0.000, C 0.000 }
gfCNCPoint2[27417] = {X 471.8007, Y 46.9091, Z -3.8333, A 0.000, B 0.000, C 0.000 }
gfCNCPoint2[27418] = {X 471.4753, Y 45.9791, Z -3.8333, A 0.000, B 0.000, C 0.000 }
gfCNCPoint2[27419] = {X 471.3650, Y 45.0000, Z -3.8333, A 0.000, B 0.000, C 0.000 }
gfCNCPoint2[27420] = {X 471.3654, Y 44.1483, Z -3.8333, A 0.000, B 0.000, C 0.000 }
gfCNCPoint2[27421] = {X 471.4638, Y 43.2816, Z -3.8333, A 0.000, B 0.000, C 0.000 }
gfCNCPoint2[27422] = {X 471.7311, Y 42.4514, Z -3.8333, A 0.000, B 0.000, C 0.000 }
gfCNCPoint2[27423] = {X 472.1570, Y 41.6903, Z -3.8333, A 0.000, B 0.000, C 0.000 }
gfCNCPoint2[27424] = {X 472.7247, Y 41.0281, Z -3.8333, A 0.000, B 0.000, C 0.000 }
gfCNCPoint2[27425] = {X 473.4118, Y 40.4909, Z -3.8333, A 0.000, B 0.000, C 0.000 }
gfCNCPoint2[27426] = {X 474.1914, Y 40.0998, Z -3.8333, A 0.000, B 0.000, C 0.000 }
gfCNCPoint2[27427] = {X 478.1277, Y 32.3948, Z -3.8333, A 0.000, B 0.000, C 0.000 }
gfCNCPoint2[27428] = {X 476.8710, Y 31.5206, Z -3.8333, A 0.000, B 0.000, C 0.000 }
gfCNCPoint2[27429] = {X 475.7410, Y 30.4879, Z -3.8333, A 0.000, B 0.000, C 0.000 }
gfCNCPoint2[27430] = {X 474.7574, Y 29.3148, Z -3.8333, A 0.000, B 0.000, C 0.000 }
gfCNCPoint2[27431] = {X 473.9377, Y 28.0220, Z -3.8333, A 0.000, B 0.000, C 0.000 }
gfCNCPoint2[27432] = {X 473.2961, Y 26.6320, Z -3.8333, A 0.000, B 0.000, C 0.000 }
gfCNCPoint2[27433] = {X 472.8439, Y 25.1695, Z -3.8333, A 0.000, B 0.000, C 0.000 }
gfCNCPoint2[27434] = {X 472.5290, Y 23.4784, Z -3.8333, A 0.000, B 0.000, C 0.000 }
gfCNCPoint2[27435] = {X 472.3882, Y 21.7639, Z -3.8333, A 0.000, B 0.000, C 0.000 }
gfCNCPoint2[27436] = {X 472.4231, Y 20.0441, Z -3.8333, A 0.000, B 0.000, C 0.000 }
gfCNCPoint2[27437] = {X 472.6333, Y 18.3368, Z -3.8333, A 0.000, B 0.000, C 0.000 }
gfCNCPoint2[27438] = {X 473.0165, Y 16.6598, Z -3.8333, A 0.000, B 0.000, C 0.000 }
gfCNCPoint2[27439] = {X 473.5628, Y 15.1347, Z -3.8333, A 0.000, B 0.000, C 0.000 }
gfCNCPoint2[27440] = {X 474.3111, Y 13.6978, Z -3.8333, A 0.000, B 0.000, C 0.000 }
gfCNCPoint2[27441] = {X 475.2475, Y 12.3757, Z -3.8333, A 0.000, B 0.000, C 0.000 }
gfCNCPoint2[27442] = {X 476.3546, Y 11.1930, Z -3.8333, A 0.000, B 0.000, C 0.000 }
gfCNCPoint2[27443] = {X 477.6120, Y 10.1715, Z -3.8333, A 0.000, B 0.000, C 0.000 }
gfCNCPoint2[27444] = {X 478.9964, Y 9.3301, Z -3.8333, A 0.000, B 0.000, C 0.000 }
gfCNCPoint2[27445] = {X 480.4822, Y 8.6843, Z -3.8333, A 0.000, B 0.000, C 0.000 }
gfCNCPoint2[27446] = {X 482.0419, Y 8.2462, Z -3.8333, A 0.000, B 0.000, C 0.000 }
gfCNCPoint2[27447] = {X 484.1467, Y 7.9181, Z -3.8333, A 0.000, B 0.000, C 0.000 }
gfCNCPoint2[27448] = {X 486.2739, Y 7.8031, Z -3.8333, A 0.000, B 0.000, C 0.000 }
gfCNCPoint2[27449] = {X 486.9707, Y 7.7909, Z -3.8333, A 0.000, B 0.000, C 0.000 }
gfCNCPoint2[27450] = {X 502.2084, Y 7.7909, Z -3.8333, A 0.000, B 0.000, C 0.000 }
gfCNCPoint2[27451] = {X 502.7400, Y 7.7951, Z -3.8333, A 0.000, B 0.000, C 0.000 }
gfCNCPoint2[27452] = {X 503.7096, Y 7.9114, Z -3.8333, A 0.000, B 0.000, C 0.000 }
gfCNCPoint2[27453] = {X 504.6294, Y 8.2396, Z -3.8333, A 0.000, B 0.000, C 0.000 }
gfCNCPoint2[27454] = {X 505.4536, Y 8.7633, Z -3.8333, A 0.000, B 0.000, C 0.000 }
gfCNCPoint2[27455] = {X 506.1414, Y 9.4566, Z -3.8333, A 0.000, B 0.000, C 0.000 }
gfCNCPoint2[27456] = {X 506.6587, Y 10.2849, Z -3.8333, A 0.000, B 0.000, C 0.000 }
gfCNCPoint2[27457] = {X 506.9797, Y 11.2072, Z -3.8333, A 0.000, B 0.000, C 0.000 }
gfCNCPoint2[27458] = {X 507.0885, Y 12.1776, Z -3.8333, A 0.000, B 0.000, C 0.000 }
gfCNCPoint2[27459] = {X 507.0883, Y 13.0233, Z -3.8333, A 0.000, B 0.000, C 0.000 }
gfCNCPoint2[27460] = {X 506.9799, Y 13.9494, Z -3.8333, A 0.000, B 0.000, C 0.000 }
gfCNCPoint2[27461] = {X 506.6789, Y 14.8318, Z -3.8333, A 0.000, B 0.000, C 0.000 }
gfCNCPoint2[27462] = {X 506.1987, Y 15.6310, Z -3.8333, A 0.000, B 0.000, C 0.000 }
gfCNCPoint2[27463] = {X 505.5609, Y 16.3111, Z -3.8333, A 0.000, B 0.000, C 0.000 }
gfCNCPoint2[27464] = {X 505.5608, Y 40.8757, Z -3.8333, A 0.000, B 0.000, C 0.000 }
gfCNCPoint2[27465] = {X 506.2055, Y 41.5648, Z -3.8333, A 0.000, B 0.000, C 0.000 }
gfCNCPoint2[27466] = {X 506.6884, Y 42.3756, Z -3.8333, A 0.000, B 0.000, C 0.000 }
gfCNCPoint2[27467] = {X 506.9873, Y 43.2707, Z -3.8333, A 0.000, B 0.000, C 0.000 }
gfCNCPoint2[27468] = {X 507.0885, Y 44.2089, Z -3.8333, A 0.000, B 0.000, C 0.000 }
gfCNCPoint2[27469] = {X 507.0885, Y 45.0000, Z -3.8333, A 0.000, B 0.000, C 0.000 }
gfCNCPoint2[27470] = {X 506.9782, Y 45.9791, Z -3.8333, A 0.000, B 0.000, C 0.000 }
gfCNCPoint2[27471] = {X 506.6528, Y 46.9091, Z -3.8333, A 0.000, B 0.000, C 0.000 }
gfCNCPoint2[27472] = {X 506.1285, Y 47.7434, Z -3.8333, A 0.000, B 0.000, C 0.000 }
gfCNCPoint2[27473] = {X 505.4318, Y 48.4401, Z -3.8333, A 0.000, B 0.000, C 0.000 }
gfCNCPoint2[27474] = {X 504.5976, Y 48.9643, Z -3.8333, A 0.000, B 0.000, C 0.000 }
gfCNCPoint2[27475] = {X 503.6676, Y 49.2897, Z -3.8333, A 0.000, B 0.000, C 0.000 }
gfCNCPoint2[27476] = {X 502.6885, Y 49.4000, Z -3.8333, A 0.000, B 0.000, C 0.000 }
gfCNCPoint2[27477] = {X 496.2450, Y 49.4000, Z -3.8333, A 0.000, B 0.000, C 0.000 }
gfCNCPoint2[27478] = {X 495.2659, Y 49.2897, Z -3.8333, A 0.000, B 0.000, C 0.000 }
gfCNCPoint2[27479] = {X 494.3359, Y 48.9643, Z -3.8333, A 0.000, B 0.000, C 0.000 }
gfCNCPoint2[27480] = {X 493.5017, Y 48.4400, Z -3.8333, A 0.000, B 0.000, C 0.000 }
gfCNCPoint2[27481] = {X 492.8050, Y 47.7433, Z -3.8333, A 0.000, B 0.000, C 0.000 }
gfCNCPoint2[27482] = {X 492.2807, Y 46.9091, Z -3.8333, A 0.000, B 0.000, C 0.000 }
gfCNCPoint2[27483] = {X 491.9553, Y 45.9791, Z -3.8333, A 0.000, B 0.000, C 0.000 }
gfCNCPoint2[27484] = {X 491.8450, Y 45.0000, Z -3.8333, A 0.000, B 0.000, C 0.000 }
gfCNCPoint2[27485] = {X 491.8454, Y 44.1483, Z -3.8333, A 0.000, B 0.000, C 0.000 }
gfCNCPoint2[27486] = {X 491.9559, Y 43.2275, Z -3.8333, A 0.000, B 0.000, C 0.000 }
gfCNCPoint2[27487] = {X 492.2568, Y 42.3503, Z -3.8333, A 0.000, B 0.000, C 0.000 }
gfCNCPoint2[27488] = {X 492.7349, Y 41.5556, Z -3.8333, A 0.000, B 0.000, C 0.000 }
gfCNCPoint2[27489] = {X 493.3690, Y 40.8789, Z -3.8333, A 0.000, B 0.000, C 0.000 }
gfCNCPoint2[27490] = {X 493.3690, Y 34.5538, Z -3.8333, A 0.000, B 0.000, C 0.000 }
gfCNCPoint2[27491] = {X 490.7730, Y 34.5538, Z -3.8333, A 0.000, B 0.000, C 0.000 }
gfCNCPoint2[27492] = {X 486.5269, Y 42.8224, Z -3.8333, A 0.000, B 0.000, C 0.000 }
gfCNCPoint2[27493] = {X 486.6946, Y 43.5066, Z -3.8333, A 0.000, B 0.000, C 0.000 }
gfCNCPoint2[27494] = {X 486.7510, Y 44.2089, Z -3.8333, A 0.000, B 0.000, C 0.000 }
gfCNCPoint2[27495] = {X 486.7510, Y 45.0000, Z -3.8333, A 0.000, B 0.000, C 0.000 }
gfCNCPoint2[27496] = {X 486.6407, Y 45.9791, Z -3.8333, A 0.000, B 0.000, C 0.000 }
gfCNCPoint2[27497] = {X 486.3153, Y 46.9091, Z -3.8333, A 0.000, B 0.000, C 0.000 }
gfCNCPoint2[27498] = {X 485.7911, Y 47.7434, Z -3.8333, A 0.000, B 0.000, C 0.000 }
gfCNCPoint2[27499] = {X 485.0944, Y 48.4401, Z -3.8333, A 0.000, B 0.000, C 0.000 }
gfCNCPoint2[27500] = {X 484.2601, Y 48.9643, Z -3.8333, A 0.000, B 0.000, C 0.000 }
gfCNCPoint2[27501] = {X 483.3301, Y 49.2897, Z -3.8333, A 0.000, B 0.000, C 0.000 }
gfCNCPoint2[27502] = {X 482.3510, Y 49.4000, Z -3.8333, A 0.000, B 0.000, C 0.000 }
gfCNCPoint2[27503] = {X 480.2695, Y 49.4000, Z -3.8333, A 0.000, B 0.000, C 0.000 }
gfCNCPoint2[27504] = {X 480.2695, Y 49.8800, Z -3.8333, A 0.000, B 0.000, C 0.000 }
gfCNCPoint2[27505] = {X 481.4067, Y 50.7435, Z -3.8333, A 0.000, B 0.000, C 0.000 }
gfCNCPoint2[27506] = {X 482.4044, Y 51.7649, Z -3.8333, A 0.000, B 0.000, C 0.000 }
gfCNCPoint2[27507] = {X 483.2411, Y 52.9219, Z -3.8333, A 0.000, B 0.000, C 0.000 }
gfCNCPoint2[27508] = {X 483.8615, Y 54.1044, Z -3.8333, A 0.000, B 0.000, C 0.000 }
gfCNCPoint2[27509] = {X 484.3133, Y 55.3610, Z -3.8333, A 0.000, B 0.000, C 0.000 }
gfCNCPoint2[27510] = {X 484.5879, Y 56.6678, Z -3.8333, A 0.000, B 0.000, C 0.000 }
gfCNCPoint2[27511] = {X 484.6800, Y 58.0000, Z -3.8333, A 0.000, B 0.000, C 0.000 }
gfCNCPoint2[27512] = {X 484.6797, Y 59.0140, Z -3.8333, A 0.000, B 0.000, C 0.000 }
gfCNCPoint2[27513] = {X 484.5592, Y 60.4585, Z -3.8333, A 0.000, B 0.000, C 0.000 }
gfCNCPoint2[27514] = {X 484.2244, Y 61.8687, Z -3.8333, A 0.000, B 0.000, C 0.000 }
gfCNCPoint2[27515] = {X 483.6828, Y 63.2132, Z -3.8333, A 0.000, B 0.000, C 0.000 }
gfCNCPoint2[27516] = {X 482.9466, Y 64.4617, Z -3.8333, A 0.000, B 0.000, C 0.000 }
gfCNCPoint2[27517] = {X 482.0321, Y 65.5863, Z -3.8333, A 0.000, B 0.000, C 0.000 }
gfCNCPoint2[27518] = {X 480.9600, Y 66.5617, Z -3.8333, A 0.000, B 0.000, C 0.000 }
gfCNCPoint2[27519] = {X 480.9604, Y 89.4445, Z -3.8333, A 0.000, B 0.000, C 0.000 }
gfCNCPoint2[27520] = {X 482.0600, Y 90.4468, Z -3.8333, A 0.000, B 0.000, C 0.000 }
gfCNCPoint2[27521] = {X 482.9925, Y 91.6061, Z -3.8333, A 0.000, B 0.000, C 0.000 }
gfCNCPoint2[27522] = {X 483.7358, Y 92.8950, Z -3.8333, A 0.000, B 0.000, C 0.000 }
gfCNCPoint2[27523] = {X 507.6816, Y 92.8950, Z -3.8333, A 0.000, B 0.000, C 0.000 }
gfCNCPoint2[27524] = {X 507.6816, Y 95.2950, Z -3.8333, A 0.000, B 0.000, C 0.000 }
gfCNCPoint2[27525] = {X 595.2965, Y 95.2950, Z -3.8333, A 0.000, B 0.000, C 0.000 }
gfCNCPoint2[27526] = {X 595.2965, Y 54.2000, Z -3.8333, A 0.000, B 0.000, C 0.000 }
gfCNCPoint2[27527] = {X 593.5565, Y 54.2000, Z -3.8333, A 0.000, B 0.000, C 0.000 }
gfCNCPoint2[27528] = {X 592.2403, Y 54.1053, Z -3.8333, A 0.000, B 0.000, C 0.000 }
gfCNCPoint2[27529] = {X 590.9511, Y 53.8233, Z -3.8333, A 0.000, B 0.000, C 0.000 }
gfCNCPoint2[27530] = {X 589.7155, Y 53.3598, Z -3.8333, A 0.000, B 0.000, C 0.000 }
gfCNCPoint2[27531] = {X 588.5589, Y 52.7242, Z -3.8333, A 0.000, B 0.000, C 0.000 }
gfCNCPoint2[27532] = {X 587.5052, Y 51.9297, Z -3.8333, A 0.000, B 0.000, C 0.000 }
gfCNCPoint2[27533] = {X 586.4956, Y 52.6955, Z -3.8333, A 0.000, B 0.000, C 0.000 }
gfCNCPoint2[27534] = {X 585.3903, Y 53.3153, Z -3.8333, A 0.000, B 0.000, C 0.000 }
gfCNCPoint2[27535] = {X 584.1375, Y 53.7999, Z -3.8333, A 0.000, B 0.000, C 0.000 }
gfCNCPoint2[27536] = {X 582.8276, Y 54.0969, Z -3.8333, A 0.000, B 0.000, C 0.000 }
gfCNCPoint2[27537] = {X 581.4884, Y 54.1999, Z -3.8333, A 0.000, B 0.000, C 0.000 }
gfCNCPoint2[27538] = {X 580.1485, Y 54.1069, Z -3.8333, A 0.000, B 0.000, C 0.000 }
gfCNCPoint2[27539] = {X 578.8364, Y 53.8198, Z -3.8333, A 0.000, B 0.000, C 0.000 }
gfCNCPoint2[27540] = {X 577.5801, Y 53.3447, Z -3.8333, A 0.000, B 0.000, C 0.000 }
gfCNCPoint2[27541] = {X 576.4063, Y 52.6917, Z -3.8333, A 0.000, B 0.000, C 0.000 }
gfCNCPoint2[27542] = {X 575.3401, Y 51.8748, Z -3.8333, A 0.000, B 0.000, C 0.000 }
gfCNCPoint2[27543] = {X 574.2798, Y 52.6879, Z -3.8333, A 0.000, B 0.000, C 0.000 }
gfCNCPoint2[27544] = {X 573.1128, Y 53.3388, Z -3.8333, A 0.000, B 0.000, C 0.000 }
gfCNCPoint2[27545] = {X 571.8638, Y 53.8139, Z -3.8333, A 0.000, B 0.000, C 0.000 }
gfCNCPoint2[27546] = {X 570.5592, Y 54.1030, Z -3.8333, A 0.000, B 0.000, C 0.000 }
gfCNCPoint2[27547] = {X 569.2264, Y 54.2000, Z -3.8333, A 0.000, B 0.000, C 0.000 }
gfCNCPoint2[27548] = {X 562.4443, Y 54.2000, Z -3.8333, A 0.000, B 0.000, C 0.000 }
gfCNCPoint2[27549] = {X 561.0051, Y 54.0867, Z -3.8333, A 0.000, B 0.000, C 0.000 }
gfCNCPoint2[27550] = {X 559.6013, Y 53.7497, Z -3.8333, A 0.000, B 0.000, C 0.000 }
gfCNCPoint2[27551] = {X 558.2676, Y 53.1973, Z -3.8333, A 0.000, B 0.000, C 0.000 }
gfCNCPoint2[27552] = {X 557.0367, Y 52.4430, Z -3.8333, A 0.000, B 0.000, C 0.000 }
gfCNCPoint2[27553] = {X 555.9389, Y 51.5054, Z -3.8333, A 0.000, B 0.000, C 0.000 }
gfCNCPoint2[27554] = {X 555.0013, Y 50.4076, Z -3.8333, A 0.000, B 0.000, C 0.000 }
gfCNCPoint2[27555] = {X 554.2470, Y 49.1767, Z -3.8333, A 0.000, B 0.000, C 0.000 }
gfCNCPoint2[27556] = {X 553.6946, Y 47.8430, Z -3.8333, A 0.000, B 0.000, C 0.000 }
gfCNCPoint2[27557] = {X 553.3576, Y 46.4392, Z -3.8333, A 0.000, B 0.000, C 0.000 }
gfCNCPoint2[27558] = {X 553.2443, Y 45.0000, Z -3.8333, A 0.000, B 0.000, C 0.000 }
gfCNCPoint2[27559] = {X 553.2444, Y 44.0430, Z -3.8333, A 0.000, B 0.000, C 0.000 }
gfCNCPoint2[27560] = {X 553.3468, Y 42.7112, Z -3.8333, A 0.000, B 0.000, C 0.000 }
gfCNCPoint2[27561] = {X 553.6403, Y 41.4081, Z -3.8333, A 0.000, B 0.000, C 0.000 }
gfCNCPoint2[27562] = {X 554.1187, Y 40.1610, Z -3.8333, A 0.000, B 0.000, C 0.000 }
gfCNCPoint2[27563] = {X 554.7721, Y 38.9959, Z -3.8333, A 0.000, B 0.000, C 0.000 }
gfCNCPoint2[27564] = {X 554.7721, Y 11.0112, Z -3.8333, A 0.000, B 0.000, C 0.000 }
gfCNCPoint2[27565] = {X 554.1220, Y 9.8556, Z -3.8333, A 0.000, B 0.000, C 0.000 }
gfCNCPoint2[27566] = {X 553.6447, Y 8.6187, Z -3.8333, A 0.000, B 0.000, C 0.000 }
gfCNCPoint2[27567] = {X 553.3502, Y 7.3259, Z -3.8333, A 0.000, B 0.000, C 0.000 }
gfCNCPoint2[27568] = {X 553.2446, Y 6.0043, Z -3.8333, A 0.000, B 0.000, C 0.000 }
gfCNCPoint2[27569] = {X 553.2443, Y 5.0000, Z -3.8333, A 0.000, B 0.000, C 0.000 }
gfCNCPoint2[27570] = {X 553.2455, Y 4.8525, Z -3.8333, A 0.000, B 0.000, C 0.000 }
gfCNCPoint2[27571] = {X 553.2490, Y 4.7050, Z -3.8333, A 0.000, B 0.000, C 0.000 }
gfCNCPoint2[27572] = {X 365.1868, Y 4.7050, Z -3.8333, A 0.000, B 0.000, C 0.000 }
